	10 : 	(************* Check Sensors Before Homing ****************)
			Station.Status 		:= 'Org10: Check Sensors Before Homing';
			Station.StatusInt	:= 120;
			
			Station.OriginRunStep 	:= 20;	

	20	:	(********** Origin Condition Check ****************)
			IF  CO_FlapGuide_Cyl_Var.S_WorkPos AND CO_Brdg_Cyl_Var.S_WorkPos AND
				(H_ER_CtnRdyForPushIn AND NOT H_ER_CtnPushInDone) THEN
				Station.OriginRunStep 		:= Station.OriginRunStep + 10;				
			ELSE
				Station.OriginRunStep 		:= 100;
			END_IF
		
	30 : 	(************* Bridge Cylinder, Flap Guides Forward ****************)
		
			CO_Brdg_Cyl_Var.In_OrgWork 		:= TRUE;
			CO_Brdg_Cyl_Var.In_OrgHome 		:= FALSE;
			CO_FlapGuide_Cyl_Var.In_OrgWork := TRUE;
			CO_FlapGuide_Cyl_Var.In_OrgHome := FALSE;
			
			CO_YPush_Srv_Var.In_PosCmd := H_CO_YPush_Srv_CtnFinalPos;
			CO_YPush_Srv_Var.In_VelCmd := A_Srv_YPusherLoSpeed;
			IF CO_YPush_Srv_Var.In_MoveXLock AND CO_Brdg_Cyl_Var.In_WorkXLock THEN
				CO_YPush_Srv_Var.In_MoveAbs := TRUE;
			END_IF
		
			IF CO_Brdg_Cyl_Var.S_WorkPos AND 
				CO_FlapGuide_Cyl_Var.S_WorkPos THEN
				CO_YPush_Srv_Var.In_MoveAbs 		:= FALSE;
				CO_Brdg_Cyl_Var.In_AutoWork 		:= FALSE;
				CO_FFlapBrdg_Cyl_Var.In_OrgWork 	:= FALSE;
				CO_FlapGuide_Cyl_Var.In_OrgWork 	:= FALSE;
				Station.OriginRunStep  				:= Station.OriginRunStep  + 10;
			END_IF		
			
	40 : 	(************* Move Y Pusher To Push Stack into Carton  ****************)	
			CO_YPush_Srv_Var.In_PosCmd := H_CO_YPush_Srv_CtnFinalPos;
			CO_YPush_Srv_Var.In_VelCmd := A_Srv_YPusherLoSpeed;
			CO_YPush_Srv_Var.In_MoveAbs := TRUE;

			IF 	CO_YPush_Srv_Var.Out_CurrPos >= (CO_YPush_Srv_Var.In_PosCmd - 100) THEN
				CO_YPush_Strk_Cyl_Var.In_OrgWork := TRUE;
				CO_YPush_Strk_Cyl_Var.In_OrgHome := FALSE;
			END_IF
			
			IF ((fcComparePos(CurrPos:= CO_YPush_Srv_Var.Out_CurrPos, TargetPos:= CO_YPush_Srv_Var.In_PosCmd, Tolerance := 0.5)) AND
							CO_YPush_Srv_Var.Out_InPos) AND
				CO_YPush_Strk_Cyl_Var.S_WorkPos THEN	
				H_CO_StkRdyForYPush 				:= FALSE;	
				H_CO_Bdl_StkY_Count 				:= 0;	
				CO_YPush_Srv_Var.In_MoveAbs 		:= FALSE;
				CO_YPush_Strk_Cyl_Var.In_OrgWork 	:= FALSE;
				Station.OriginRunStep 				:= 50;
				
				IF NOT Cfg_BypassErector AND H_ER_CtnRdyForPushIn THEN
					H_ER_CtnPushInDone := TRUE;
				END_IF
					H_ER_CtnRdyForPushIn := FALSE;
				
			END_IF
			
	50 : 	(************* push into box  after y push  ****************)
			Station.Status 		:= '120: Push into box';
			Station.StatusInt	:= 151;
			
			CO_YPush_Cyl_Var.In_OrgWork := TRUE;
			CO_YPush_Cyl_Var.In_OrgHome := FALSE;
			
			IF  CO_YPush_Cyl_Var.S_HomePos THEN
				CO_YPush_Cyl_Var.In_AutoWork := TRUE;
				CO_YPush_Cyl_Var.In_AutoHome := FALSE;			
				CO_YPush_Srv_Var.In_MoveAbs := FALSE; 
				Station.RunStep := 100;			
			END_IF
			
	
			
	100 : 	(************* Y Pusher Servo Move to Safe Pos ****************)
			Station.Status 		:= 'Org30: Y Pusher Servo Move to Safe Pos ';
			Station.StatusInt	:= 172;
			CO_YPush_Strk_Cyl_Var.In_OrgHome 	:= NOT CO_YPush_Strk_Cyl_Var.S_HomePos;	
			
		IF CO_YPush_Srv_Var.Out_CurrPos > H_CO_YPush_Srv_SafePosition THEN
			CO_YPush_Srv_Var.In_PosCmd := H_CO_YPush_Srv_SafePosition; 
			CO_YPush_Srv_Var.In_VelCmd := A_Srv_BeltAutoHiSpeed;
			CO_YPush_Srv_Var.In_MoveAbs := TRUE;
		ELSE
			CO_YPush_Srv_Var.In_MoveAbs := FALSE;
			Station.OriginRunStep := Station.OriginRunStep+5;	
		END_IF
				
			IF ((fcComparePos(CurrPos:= CO_YPush_Srv_Var.Out_CurrPos, TargetPos:= H_CO_YPush_Srv_SafePosition,  Tolerance := 0.5)) AND
				CO_YPush_Srv_Var.Out_InPos) THEN
				CO_YPush_Srv_Var.In_MoveAbs := FALSE;
				Station.OriginRunStep := Station.OriginRunStep+5;	
			END_IF
			
	105:	(************* Y Pusher Servo Move to Standby Pos ****************)			
			CO_YPush_Cyl_Var.In_OrgWork := TRUE;
			CO_YPush_Cyl_Var.In_OrgHome := FALSE;
			
			IF CO_YPush_Cyl_Var.S_WorkPos THEN
				CO_YPush_Srv_Var.In_PosCmd := H_CO_YPush_Srv_CurrStandbyPos; 
				CO_YPush_Srv_Var.In_VelCmd := A_Srv_BeltAutoHiSpeed;
				CO_YPush_Srv_Var.In_MoveAbs := TRUE;
			END_IF
			
			IF ((fcComparePos(CurrPos:= CO_YPush_Srv_Var.Out_CurrPos, TargetPos:= H_CO_YPush_Srv_CurrStandbyPos, Tolerance := 0.5)) AND
							CO_YPush_Srv_Var.Out_InPos) THEN
				CO_YPush_Srv_Var.In_MoveAbs := FALSE;
			Station.OriginRunStep := Station.OriginRunStep+5;	
			END_IF
			
	110 : 	(************* All Cylinders Home ****************)
			Station.Status 		:= 'Org40: All Cylinders Home';
			Station.StatusInt	:= 173;
			
			
			CO_Brdg_Cyl_Var.In_OrgHome 			:= NOT CO_Brdg_Cyl_Var.S_HomePos;
			CO_Brdg_Cyl_Var.In_OrgWORK			:= FALSE;	
			CO_FlapGuide_Cyl_Var.In_OrgHome 	:= NOT CO_FlapGuide_Cyl_Var.S_HomePos;				
			CO_YPush_Cyl_Var.In_OrgWork 		:= FALSE;
			CO_YPush_Cyl_Var.In_OrgHome 		:= TRUE;


			IF  CO_YPush_Strk_Cyl_Var.S_HomePos AND
				CO_Brdg_Cyl_Var.S_HomePos 		AND
				CO_FlapGuide_Cyl_Var.S_HomePos 	AND
				CO_YPush_Cyl_Var.S_HomePos		THEN
				CO_YPush_Strk_Cyl_Var.In_OrgHome 	:= FALSE;	
				CO_Brdg_Cyl_Var.In_OrgHome 			:= FALSE;	
				CO_FlapGuide_Cyl_Var.In_OrgHome 	:= FALSE;
				CO_YPush_Cyl_Var.In_OrgWork 		:= FALSE;
				CO_YPush_Cyl_Var.In_OrgHome 		:= FALSE;

				IF CO_YPush_WA_Origin THEN
					Station.OriginRunStep := 0;	
				END_IF	
			END_IF
		


					
	END_CASE

ELSE

	Station.OriginRunStep := 0;	
	
END_IF

END_PROGRAM

// ---- POUs/Collator/CO_Cylinder_Output.TcPOU
PROGRAM CO_Cylinder_Output
VAR
	Reset:BOOL;
	bEnable:BOOL;
	CO_Brdg_Cyl_Home_Tmr : TON;
	CO_Brdg_Cyl_Work_Tmr : TON;
	
END_VAR

bEnable := NOT MC.Trouble;

(*Refer to FastTask Folder for Stack Release Cylinder Control*)

CO_Brdg_Cyl_Var.In_HomeXLock := TRUE;
CO_Brdg_Cyl_Var.In_WorkXLock := (NOT ER_Arm_Srv_Var.Out_Busy OR NOT ER_Arm_Vac_Var.S_Vacuum) AND
								ER_RFlapL_Cyl_Var.S_HomePos;
CO_Brdg_Cyl_Home_Tmr(IN:= O_CO_Brdg_Bwd, PT := T#2S);
CO_Brdg_Cyl_Work_Tmr(IN:= O_CO_Brdg_Fwd, PT := T#2S);

CO_Brdg_Cyl(				
	IN_CylName		:='3Y3 PUSHER BRIDGE', 	
	In_Enable		:= bEnable, 	
	In_Reset		:= MC.ResetPressed, 	
	In_WorkRS		:= I_CO_Brdg_Fwd, 	
	In_HomeRS		:= I_CO_Brdg_Bwd, 	
	In_WorkTON		:= T#10MS, 	
	In_HomeTON		:= T#10MS, 	
	in_Timeout		:= TP_Cyl_Timeout, 	
	Out_WorkSV		=> O_CO_Brdg_Fwd, 	
	Out_HomeSV		=> O_CO_Brdg_Bwd, 	
	CylVar			:= CO_Brdg_Cyl_Var,
	Station			:= SC[2]);

CO_FlapGuide_Cyl_Var.In_HomeXLock := TRUE;
CO_FlapGuide_Cyl_Var.In_WorkXLock := TRUE;

CO_FlapGuide_Cyl(				
	IN_CylName		:='3Y4/5 PUSHER FLAP GUIDE', 	
	In_Enable		:= bEnable, 	
	In_Reset		:= MC.ResetPressed, 	
	In_WorkRS		:= I_CO_RFlapGuide_Fwd AND I_CO_FFlapGuide_Fwd, 	
	In_HomeRS		:= I_CO_RFlapGuide_Bwd AND I_CO_FFlapGuide_Bwd, 	
	In_WorkTON		:= T#10MS, 	
	In_HomeTON		:= T#10MS, 	
	in_Timeout		:= TP_Cyl_Timeout, 	
	Out_WorkSV		=> O_CO_RFlapGuide_Fwd, 	
	Out_HomeSV		=> O_CO_RFlapGuide_Bwd, 	
	CylVar			:= CO_FlapGuide_Cyl_Var,
	Station			:= SC[2]);

	O_CO_FFlapBrdg_Fwd:=O_CO_RFlapGuide_Fwd;
	O_CO_FFlapBrdg_Bwd:=O_CO_RFlapGuide_Bwd;
	
CO_YPush_Strk_Cyl_Var.In_HomeXLock := TRUE;
CO_YPush_Strk_Cyl_Var.In_WorkXLock := CO_YPush_Cyl_Var.S_HomePos;

CO_YPush_Strk_Cyl(				
	IN_CylName		:='3Y2 Y PUSHER STROKE', 	
	In_Enable		:= bEnable, 	
	In_Reset		:= MC.ResetPressed, 	
	In_WorkRS		:= I_CO_YPush_Strk_Fwd, 	
	In_HomeRS		:= I_CO_YPush_Strk_Bwd, 	
	In_WorkTON		:= T#10MS, 	
	In_HomeTON		:= T#10MS, 	
	in_Timeout		:= TP_Cyl_Timeout, 	
	Out_WorkSV		=> O_CO_YPush_Strk_Fwd, 	
	Out_HomeSV		=> O_CO_YPush_Strk_Bwd, 	
	CylVar			:= CO_YPush_Strk_Cyl_Var,
	Station			:= SC[2]);

CO_YPush_Cyl_Var.In_HomeXLock := TRUE ;
CO_YPush_Cyl_Var.In_WorkXLock := CO_YPush_Srv_Var.Out_CurrPos <= H_CO_YPush_Srv_SafePosition + 1 ;

CO_YPush_Cyl(				
	IN_CylName		:='3Y1 Y PUSHER', 	
	In_Enable		:= bEnable, 	
	In_Reset		:= MC.ResetPressed, 	
	In_WorkRS		:= I_CO_YPush_Up, 	
	In_HomeRS		:= I_CO_YPush_Dn, 	
	In_WorkTON		:= T#10MS, 	
	In_HomeTON		:= T#10MS, 	
	in_Timeout		:= TP_Cyl_Timeout, 	
	Out_WorkSV		=> O_CO_YPush_Up, 	
	Out_HomeSV		=> O_CO_YPush_Dn, 	
	CylVar			:= CO_YPush_Cyl_Var,
Station			:= SC[2]);

CO_PalletLoc_Cyl_Var.In_HomeXLock := TRUE;
CO_PalletLoc_Cyl_Var.In_WorkXLock := TRUE;
	
CO_PalletLoc_Cyl(				
	IN_CylName		:='3Y2 Y PALLET LOCATING', 	
	In_Enable		:= bEnable, 	
	In_Reset		:= MC.ResetPressed, 	
	In_WorkRS		:= I_CO_PalletLocating_Fwd, 	
	In_HomeRS		:= I_CO_PalletLocating_Bwd, 	
	In_WorkTON		:= T#10MS, 	
	In_HomeTON		:= T#10MS, 	
	in_Timeout		:= TP_Cyl_Timeout, 	
	Out_WorkSV		=> O_CO_PalletLocating_Fwd, 	
	Out_HomeSV		=> O_CO_PalletLocating_Bwd, 	
	CylVar			:= CO_PalletLoc_Cyl_Var,
	Station			:= SC[2]);

CO_Sing1_Cyl_Var.In_HomeXLock := TRUE;
CO_Sing1_Cyl_Var.In_WorkXLock := TRUE;
CO_Sing1_Cyl(				
	IN_CylName		:='3Y2 Singulator 1', 	
	In_Enable		:= bEnable, 	
	In_Reset		:= MC.ResetPressed, 	
	In_WorkRS		:= I_CO_Sing1_Fwd, 	
	In_HomeRS		:= I_CO_Sing1_Bwd, 	
	In_WorkTON		:= T#10MS, 	
	In_HomeTON		:= T#10MS, 	
	in_Timeout		:= TP_Cyl_Timeout, 	
	Out_WorkSV		=> O_CO_Sing1_Fwd, 	
	Out_HomeSV		=> O_CO_Sing1_Bwd, 	
	CylVar			:= CO_Sing1_Cyl_Var,
	Station			:= SC[2]);

CO_Sing2_Cyl_Var.In_HomeXLock := TRUE;
CO_Sing2_Cyl_Var.In_WorkXLock := TRUE;	
CO_Sing2_Cyl(				
	IN_CylName		:='3Y2 Singulator 1', 	
	In_Enable		:= bEnable, 	
	In_Reset		:= MC.ResetPressed, 	
	In_WorkRS		:= I_CO_Sing2_Fwd, 	
	In_HomeRS		:= I_CO_Sing2_Bwd, 	
	In_WorkTON		:= T#10MS, 	
	In_HomeTON		:= T#10MS, 	
	in_Timeout		:= TP_Cyl_Timeout, 	
	Out_WorkSV		=> O_CO_Sing2_Fwd, 	
	Out_HomeSV		=> O_CO_Sing2_Bwd, 	
	CylVar			:= CO_Sing2_Cyl_Var,
	Station			:= SC[2]);

END_PROGRAM

// ---- POUs/Collator/CO_Servo_Output.TcPOU
PROGRAM CO_Servo_Output
VAR
	Reset:BOOL;
	plsStopMove: R_trig;
	bEnable: BOOL;
	bEnable_Stack: BOOL;
	bEnable_XPush: BOOL;
	bEnable_YPush: BOOL;
END_VAR

IF (MC.AutoMode OR SC[1].M_Step OR SC[2].M_Step) AND NOT CO.Bypass THEN
	CO_YPush_Srv_Var.In_ServoOn := TRUE;
END_IF

IF CO.OriginSchRun OR MC.OriginSchRun or mc.AutoMode or (mc.ResetPressed AND NOT mc.Trouble) THEN
	CO_YPush_Srv_Var.In_ServoOn := TRUE;
END_IF

 
bEnable_Stack := NOT (CO_Stack.MajorFault OR CO_Stack.MinorFault OR CO_Stack.DeviceFault OR MC.Trouble);
bEnable_YPush := NOT (CO_YPush.MajorFault OR CO_YPush.MinorFault OR CO_YPush.DeviceFault OR MC.Trouble);


(*CO_M5 Collator Y Pusher Motor - 111M1*)

IF Cfg_CollDircLtoR THEN
CO_YPush_Srv_Var.In_MoveXLock := 	((CO_FlapGuide_Cyl_Var.S_WorkPos AND
										ER_FFlapL_Cyl_Var.S_HomePos AND
										ER_RFlapL_Cyl_Var.S_HomePos) OR
									(CO_YPush_Srv_Var.Out_CurrPos <= H_CO_YPush_Srv_CtnFinalPos+200)) ;
ELSE
CO_YPush_Srv_Var.In_MoveXLock := 	((CO_FlapGuide_Cyl_Var.S_WorkPos AND
										ER_FFlapR_Cyl_Var.S_HomePos AND
										ER_RFlapR_Cyl_Var.S_HomePos) OR
									(CO_YPush_Srv_Var.Out_CurrPos <= H_CO_YPush_Srv_CtnFinalPos+200));
END_IF
CO_YPush_Srv_Drive(
	In_Enable:= bEnable_YPush, 
	In_Reset := MC.ResetPressed,
	In_AbsEncoder:= TRUE, 
	In_DriveInput:= CO_YPush_Srv_Input, 
	In_CommState:= CO_YPush_Srv_State, 
	Out_DriveOutput=> CO_YPush_Srv_Output, 
	Out_DriveFeedRateOverride=> CO_YPush_Srv_Feedrate, 
	DriveVar:= CO_YPush_Srv_Var,
	Station			:= SC[2]);

IF mc.ManualMode THEN	
	CO_YPush_Srv_Feedrate := 10000;
ELSE
	CO_YPush_Srv_Feedrate :=    INT_TO_UINT(hmi.V_MachineSpeed * 100);
END_IF

END_PROGRAM

// ---- POUs/Collator/CO_Nordson.TcPOU
PROGRAM CO_Nordson
VAR
	PumpOnOff	: fbOnOffDevCtrl;
	Standby		: fbOnOffDevCtrl;
	HeaterOn	: fbOnOffDevCtrl;
END_VAR



PumpOnOff(
	IN_DevName:= 'Pump OnOff', 
	In_Enable:= TRUE, 
	In_Reset:= MC.ResetPressed, 
	In_AutoON:= ER_Nordson_PumpOnOff_Var.In_AutoON , 
	In_OrgON:= ER_Nordson_PumpOnOff_Var.In_OrgOn , 
	In_OnXLock:= TRUE, 
	In_ONSig:=PumpOnOff.Out_OnSV , 
	In_OnTON:= , 
	in_Timeout:= T#1S, 
	Out_OnSV=> O_Nord_Auto , 
	E_OnErr=> , 
	S_OnSig=> );
	
Standby(
	IN_DevName:= 'Standby', 
	In_Enable:= TRUE, 
	In_Reset:= MC.ResetPressed, 
	In_AutoON:= ER_Nordson_Standby_Var.In_AutoON , 
	In_OrgON:= ER_Nordson_Standby_Var.In_OrgOn, 
	In_OnXLock:= TRUE , 
	In_ONSig:= Standby.Out_OnSV, 
	In_OnTON:= , 
	in_Timeout:= T#1S, 
	Out_OnSV=> O_Nord_Standby , 
	E_OnErr=> , 
	S_OnSig=> );	
	
HeaterOn(
	IN_DevName:= 'Heater On', 
	In_Enable:= TRUE, 
	In_Reset:= MC.ResetPressed, 
	In_AutoON:= ER_Nordson_HeaterOn_Var.In_AutoON  , 
	In_OrgON:= ER_Nordson_HeaterOn_Var.In_OrgOn, 
	In_OnXLock:= TRUE , 
	In_ONSig:= HeaterOn.Out_OnSV, 
	In_OnTON:= , 
	in_Timeout:= T#1S, 
	Out_OnSV=> O_Nord_HeaterOn , 
	E_OnErr=> , 
	S_OnSig=> );

END_PROGRAM

// ---- POUs/FB/fbOnOffDevCtrl.TcPOU
FUNCTION_BLOCK fbOnOffDevCtrl

VAR_INPUT
	IN:BOOL;
	IN_DevName:STRING;
	In_Enable:BOOL;
	In_Reset:BOOL;


	(*Trigger*)
	In_AutoON:BOOL;
	In_OrgON:BOOL;

	(*Mechanical Interlock*)
	In_OnXLock:BOOL;

	(*Sensors*)
	In_ONSig:BOOL;

	(*Timer*)
	In_OnTON:TIME;
	in_Timeout:TIME;

END_VAR

VAR_OUTPUT
	Q:BOOL;
	Out_OnSV:BOOL;
	E_OnErr:BOOL;
	S_OnSig:BOOL;

END_VAR

VAR_IN_OUT
	
END_VAR

VAR

	(* Trigger*)
	T_ManOn:BOOL;
	T_ManOff:BOOL;

	Loc_On:BOOL;
	On_TOut: TON;
	On_TON: TON;
	Loc_OnPls: BOOL;
	OnPls: R_TRIG;
	Out_RSErr:BOOL;
	OnPosPls: F_TRIG;

END_VAR
VAR_IN_OUT

END_VAR
VAR // added by the converter: edge detectors and wires of the graphical bodies
    _w1 : BOOL;
END_VAR

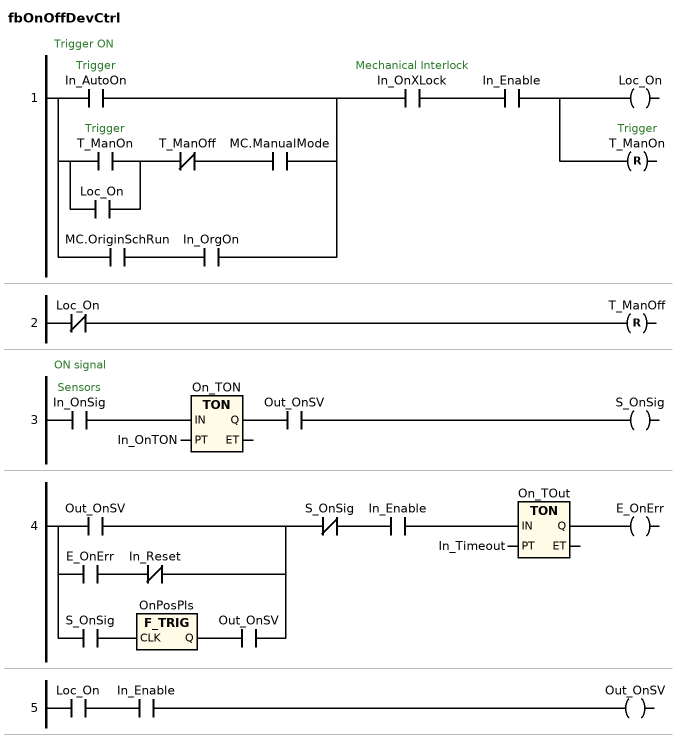
// NETWORK 1
// Trigger ON
//   In_AutoOn: Trigger
//   T_ManOn: Trigger
//   In_OnXLock: Mechanical Interlock
_w1 := (In_AutoOn OR (T_ManOn OR Loc_On) AND NOT T_ManOff AND MC.ManualMode OR MC.OriginSchRun AND In_OrgOn) AND In_OnXLock AND In_Enable;
Loc_On := _w1;
T_ManOn R= _w1;

// NETWORK 2
T_ManOff R= NOT Loc_On;

// NETWORK 3
// ON signal
//   In_OnSig: Sensors
//   In_OnTON: Timer
On_TON(IN := In_OnSig, PT := In_OnTON); // TON
S_OnSig := On_TON.Q AND Out_OnSV;

// NETWORK 4
OnPosPls(CLK := S_OnSig); // F_TRIG
On_TOut(IN := (Out_OnSV OR E_OnErr AND NOT In_Reset OR OnPosPls.Q AND Out_OnSV) AND NOT S_OnSig AND In_Enable, PT := In_Timeout); // TON
E_OnErr := On_TOut.Q;

// NETWORK 5
Out_OnSV := Loc_On AND In_Enable;

END_FUNCTION_BLOCK

// ---- POUs/Erector/ER_Main.TcPOU
PROGRAM ER_Main
VAR
END_VAR

IF Cfg_BypassErector THEN
	HMI.T_Station_BypassP[3] := TRUE;
ELSE
	HMI.T_Station_BypassP[3] := FALSE;
END_IF

ER_Timers();

ER_Error			(Station:= SC[3]);
ER_Auto_Arm			(Station:= SC[3]);
ER_Auto_FixedFlap	(Station:= SC[3]);
ER_Glue				(Station:= SC[3]);
ER_Origin			(Station:= SC[3]);

ER_Cylinder_Output();
ER_Servo_Output();
ER_Motor_Output();
ER_Vacuum_Output();

(* ER Structure is only for displaying on HMI*)
SC[3].T_OriginSearch := ER.T_OriginSearch;
ER := SC[3];

(*debug*)

IF T_SimPushIn THEN
	H_ER_CtnRdyForPushIn := FALSE;
	H_ER_CtnPushInDone := TRUE;
	H_ER_CtnSideFlapDone := FALSE;
END_IF

END_PROGRAM

// ---- POUs/Erector/ER_Timers.TcPOU
PROGRAM ER_Timers
VAR
	ER_Carton_TON	:ton;
	
END_VAR


ER_BufCv_Ctn_TON 	(IN := 	I_ER_RefillL_PE AND 
							I_ER_EmptyL_PE	AND
							I_ER_EmptyR_PE	AND
							I_ER_BufferL_PE	AND
							I_ER_BufferR_PE, pt := T#0.5S);
ER_Carton_TON(IN := 		I_ER_EmptyL_PE	AND
							I_ER_EmptyR_PE	AND
							I_ER_BufferL_PE	AND
							I_ER_BufferR_PE, pt := T#1S); 
							
ER_BufCvL_Ctn_TON 	(IN := (I_ER_EmptyL_PE AND mc.AutoRunning) OR I_ER_BufferL_PE , pt := T#70MS);
ER_BufCvR_Ctn_TON 	(IN := (I_ER_EmptyR_PE AND mc.AutoRunning) OR I_ER_BufferR_PE , pt := T#70MS);

END_PROGRAM

// ---- POUs/Erector/ER_Error.TcPOU
PROGRAM ER_Error
VAR_IN_OUT
	Station		:structStationCtrl;
END_VAR

VAR
	CaseBufferWaitTON			:Ton;
	CaseBufferEmpty_ResetTON	:ton;
	GlueEmpty_ResetTON			:ton;
	CaseBufferEmptySen_Timeout	:ton;

END_VAR

IF MC.ResetPressed THEN
	Station.SeqFaultWord := 0;
END_IF

(* 	Reserved Station.SeqFaultWord 
	= 1~49 for Major Fault
	= 100~149 for Origin Sequence Fault
	= 150~199 for Origin Width Adjust Sequence Fault
	= 200~299 for Auto Sequence Fault
	= 300~399 for misc fault listed on this page*)

Station.MajorFault := ((Station.SeqFaultWord > 0) 	AND (Station.SeqFaultWord < 50)) OR E_Case_Infeed_Safety_NOk ;
Station.MinorFault := (Station.SeqFaultWord >= 100) OR Station.DeviceFault 
													OR E_Nordson_Alarm 
													OR E_CaseBufferAlignment_Err
													OR ((E_ER_EmptyL_PE
													OR E_ER_BufferL_PE
													OR E_ER_EmptyR_PE
													OR E_ER_BufferR_PE) AND sc[3].RunStep = 0);
									
													
(* Case Infeed safety not OK *)
IF NOT I_Case_Infeed_Safety_Ok AND I_Emg_SC_OK AND I_Door_SC_OK AND NOT MC_WA_Run AND NOT Erector_SafetySensorBypass THEN
	E_Case_Infeed_Safety_NOk	:= TRUE;
END_IF

(* Case Buffer Error *)
CaseBufferWaitTON			(IN:= ((I_ER_EmptyL_PE AND NOT I_ER_BufferL_PE) OR (I_ER_EmptyR_PE AND NOT I_ER_BufferR_PE)) AND mc.AutoRunning AND (sc[3].RunStep = 0), PT:= T#30S); 
IF CaseBufferWaitTON.Q THEN
	E_CaseBufferAlignment_Err	:= TRUE;
END_IF
(*
W_CaseBuffer_is_Empty	:= 	(CaseBufferEmptying_Counter >= CaseBufferEmptying_Setting);
CaseBufferEmpty_ResetTON	( IN:= I_ER_RefillL_PE, pt:= T#3S);
IF CaseBufferEmpty_ResetTON.Q THEN
	CaseBufferEmptying_Counter	:= 0;
END_IF
*)
CaseBufferEmptySen_Timeout	( IN:= (I_ER_EmptyL_PE AND NOT I_ER_EmptyR_PE) OR (I_ER_EmptyR_PE AND NOT I_ER_EmptyL_PE), pt:= T#10S);
IF CaseBufferEmptySen_Timeout.Q THEN
	E_CaseBuffer_EmptySensors	:= TRUE;
END_IF


(*Refill Carton Buffer Warning*)
W_ER_BufRefill		:= MC.AutoMode AND NOT Station.Bypass AND 
						NOT I_ER_RefillL_PE AND NOT HMI.T_EndProd;



(* Glue Alarm/Warning *)
(*E_Nordson_Alarm		:= (NOT I_Nord_Rdy AND T_GlueEnable) AND NOT mc.DryRun AND mc.AutoRunning;*)
W_Glue_Low_Level	:= I_Nord_TankLow;
W_Glue_is_Empty		:= (GlueEmptying_Counter >= GlueEmptying_Setting );
IF NOT I_Nord_TankLow THEN 
	GlueEmptying_Counter	:= 0;
END_IF

END_PROGRAM

// ---- POUs/Erector/ER_Auto_Arm.TcPOU
                                                                                                                                                                                                                                                                                                      PROGRAM ER_Auto_Arm
VAR_IN_OUT
	Station		:structStationCtrl;
END_VAR
VAR
	tmrDelayBFlapUp:ton;
	Timeout					:TON;	
	StpCtnPE_TOFF			:Ton;
	ManualInit_TOn			:Ton;
	tmrDelayVacHold			:ton;
	CaseSupply_L_Timeout	:TON;
	CaseSupply_R_Timeout	:TON;
	tmr_Case_Buffer			:ton;	
	tmr_ArmTiltDly			:Ton;
	ServoTargetPos			:REAL;
	TimeoutTrigger			:BOOL;
	TimeoutSetting			:TIME;
	NoWPonErector			:BOOL;
	NoWPonExit				:BOOL;
	CartonPreAtStopper		:BOOL;
	GlueStart1 				:BOOL;
	GlueStart2 				:BOOL;
	DistanceAdvanceForGlue	:REAL;
	End_Production			:BOOL;	
	Case_Not_Ready 			:BOOL;	
	CaseSupply_L_TimeoutM	:BOOL;
	CaseSupply_R_TimeoutM	:BOOL;
			
END_VAR

NoWPonErector := 	NOT H_ER_CtnRdyForPushIn AND 
					NOT I_ER_StpL_Ctn_PE AND
					NOT I_ER_StpR_Ctn_PE;
							
NoWPonExit := 	NOT H_ER_CtnRdyForGlue AND
				NOT H_ER_CtnGlueDone AND
				NOT I_EX_Cv_Ctn_PE;

tmr_Case_Buffer	(IN := NOT ER_BufCv_Ctn_TON.Q AND 
					NOT (MC.DryRun  OR  End_Production ) AND
					mc.AutoRunning, pt := T#3S);			
Case_Not_Ready := 	(tmr_Case_Buffer.Q AND NOT mc.DryRun) OR 
					(NOT I_Case_Infeed_Safety_Ok AND NOT mc.E_EmgStop AND NOT mc.E_SafetyDoorOpen);
					
					
sc[3].Warning			:= Case_Not_Ready;
				
(**************************************************************************************************************)
(*	Initial Device	*)
(**************************************************************************************************************)
ManualInit_TOn (in:= mc.ManualMode AND NOT mc.OriginSchRun, pt:= T#1S);

IF mc.ManualMode AND NOT mc.OriginSchRun AND NOT ManualInit_TOn.Q THEN
	ER_Arm_Srv_Var.In_MoveAbs 			:= FALSE;
	ER_WA_Srv_Var.In_MoveAbs 			:= FALSE;	
	EX_HeightL_WA_Srv_Var.In_MoveAbs	:= FALSE;
	EX_HeightR_WA_Srv_Var.In_MoveAbs	:= FALSE;
END_IF
				
(**************************************************************************************************************)
(* GENERAL STATION MAPPING  *)
(**************************************************************************************************************)
Station.Name			:=	'CARTON ERECTOR & SIDE FLAP CLOSING';
Station.Rdy 			:= 	Station.Origin AND ER_Origin.ER_WA_Origin;
Station.AutoRun 		:=	(MC.AutoRunning OR Station.M_Step) AND 
							NOT (Station.Bypass OR Station.MajorFault OR Station.MinorFault);
Station.RunReq			:= 	(
							((NOT I_EX_Cv_Ctn_PE OR NoWPonErector) AND NoWPonErector AND NOT End_Production ) OR
							(H_ER_CtnSideFlapDone AND NoWPonExit)
							) AND
							(er_tIMERS.ER_Carton_TON.Q OR MC.DryRun OR 
							(End_Production AND (I_ER_StpL_Ctn_PE OR I_ER_StpR_Ctn_PE)) 
							);											
Station.RunCond			:=	(NOT CO_YPush.Running OR CO_YPush.RunStep >= 200) AND	(*Y Pusher Not Running Forward*) 
							( (I_Nord_Rdy and not W_Glue_is_Empty and not W_CaseBuffer_is_Empty)  OR NOT T_GlueEnable OR mc.DryRun) AND
							((NOT EX.Running OR										(*Hot Glue and Weight Check Not Running*) 	
							NoWPonErector)) AND
							NOT Station.Running AND									(*Fixed Flap Closing Not Running*)
							NOT (Station.Done OR MC.StopPressed);
Station.Run_NextStepPls	:=	(Station.AutoRun AND NOT Station.M_Step) OR 
							(Station.M_Step AND M_StepFwdPls) OR HMI.T_OneCycleRun;
Station.Run_PrevStepPls	:=	(Station.M_Step AND M_StepBwdPls);

(**************************************************************************************************************)
(* Auto Sequance*)
(**************************************************************************************************************)

Timeout(IN:=TimeoutTrigger, PT:=TimeoutSetting);
IF Timeout.Q THEN
	TimeoutTrigger := FALSE;
END_IF


tmrDelayVacHold	(IN:=Station.RunStep=30, PT:=T#0S);
tmr_ArmTiltDly	(IN:=Station.RunStep=20 AND ER_ArmTilt_Cyl_Var.S_HomePos, pt:= T#0.2S);
 
(********************* Case Supply Sequence Start ********************************)
	CaseSupply_L_Timeout	(IN:= ER_BufCvL_Mtr_Var.S_Running, PT:= T#60S);
	CaseSupply_R_Timeout	(IN:= ER_BufCvR_Mtr_Var.S_Running, PT:= T#60S);
	
	IF CaseSupply_L_Timeout.q THEN
		CaseSupply_L_TimeoutM	:= TRUE;
	END_IF
	IF CaseSupply_R_Timeout.q THEN
		CaseSupply_R_TimeoutM	:= TRUE;
	END_IF
	IF I_ER_RefillL_PE OR NOT mc.AutoRunning THEN
		CaseSupply_L_TimeoutM	:= FALSE;
		CaseSupply_R_TimeoutM	:= FALSE;
	END_IF
		
	ER_BufCvL_Mtr_Var.In_AutoON := NOT  ER_BufCvL_Ctn_TON.Q AND NOT CaseSupply_L_TimeoutM AND NOT(STation.RunStep >= 20 AND Station.RunStep <40)  ;
	ER_BufCvR_Mtr_Var.In_AutoON := NOT  ER_BufCvR_Ctn_TON.Q AND	NOT CaseSupply_L_TimeoutM AND NOT(STation.RunStep >= 20 AND Station.RunStep <40)  ;	


IF Station.AutoRun OR Station.M_Step THEN

(**************************************************************************)
	CASE Station.RunStep OF

	0 : 	(************* Ready To Run ****************)
			End_Production := hmi.T_EndProd;
			
			IF Station.RunCond AND Station.RunReq AND Station.Rdy  AND
				(NOT H_ER_CtnPushInDone OR H_ER_CtnSideFlapDone)  THEN
				Station.RunStep := Station.RunStep + 5;
			ELSIF NOT Station.RunCond THEN
				Station.Status 		:= '0: Station Waiting for Run Conditions';
				Station.StatusInt	:= 1;
			ELSIF NOT Station.RunReq THEN
				Station.Status 		:= '0: Station Waiting for Run Request';
				Station.StatusInt	:= 2;
			ELSE
				Station.Status 		:= '0: Station Not Ready';
				Station.StatusInt	:= 3;
			END_IF

	5 : 	(************* Stopper Down ****************)
			(************* Case Guide Down ****************)
			Station.Status 		:= '5: Stopper & Case Guide Down';
			Station.StatusInt	:= 251;
			
			ER_StpR_Cyl_Var.In_AutoWork 		:= FALSE;
			ER_StpR_Cyl_Var.In_AutoHome 		:= TRUE;
			ER_StpL_Cyl_Var.In_AutoWork 		:= FALSE;
			ER_StpL_Cyl_Var.In_AutoHome 		:= TRUE;
			ER_CaseGuideL_Cyl_Var.In_AutoWork 	:= FALSE;
			ER_CaseGuideL_Cyl_Var.In_AutoHome 	:= TRUE;
			ER_CaseGuideR_Cyl_Var.In_AutoWork 	:= FALSE;
			ER_CaseGuideR_Cyl_Var.In_AutoHome 	:= TRUE;
			

			IF 	ER_StpR_Cyl_Var.S_HomePos AND 
				ER_StpL_Cyl_Var.S_HomePos AND
				ER_CaseGuideL_Cyl_Var.S_HomePos AND
				ER_CaseGuideR_Cyl_Var.S_HomePos AND
				Station.Run_NextStepPls THEN
				ER_StpR_Cyl_Var.In_AutoWork := FALSE;
				ER_StpL_Cyl_Var.In_AutoWork := FALSE;
				H_ER_CtnErected				:= FALSE;
				IF NOT End_Production THEN
					Station.RunStep := Station.RunStep + 5;	
				ELSE
					Station.RunStep := 30;
				END_IF
			END_IF
			
	10 : 	(************* Erector Arm Servo Move forward while Vacuum ON ****************)
			Station.Status 		:= '10: Erector Arm Servo Move Forward';
			Station.StatusInt	:= 252;
			
			IF NOT MC.DryRun  THEN
				ER_Arm_Vac_Var.In_AutoVacuum := TRUE;
				ER_Arm_Vac_Var.In_AutoPurge := FALSE;
			END_IF

			ER_Arm_Srv_Var.In_PosCmd := H_ER_Arm_Srv_CtnVacuumPos + 45;
			ER_Arm_Srv_Var.In_VelCmd := A_Srv_ErectorArmHiSpeed;
			ER_Arm_Srv_Var.In_MoveAbs := TRUE;
			
			IF H_ER_CtnSideFlapDone THEN
				ER_RFlapL_Cyl_Var.In_AutoWork := TRUE;
				ER_RFlapR_Cyl_Var.In_AutoWork := TRUE;
			END_IF
			
			IF fcComparePos(CurrPos:= ER_Arm_Srv_Var.Out_CurrPos, TargetPos:= ER_Arm_Srv_Var.In_PosCmd,5) AND
				((ER_RFlapL_Cyl_Var.S_WorkPos AND ER_RFlapR_Cyl_Var.S_WorkPos) OR
					NOT H_ER_CtnSideFlapDone) AND
					(ER_Arm_Vac_Var.S_Vacuum OR MC.DryRun) AND
				Station.Run_NextStepPls THEN				
				ER_Arm_Srv_Var.In_MoveAbs := FALSE;
				ER_Arm_Vac_Var.In_AutoVacuum := FALSE;
				Station.RunStep := Station.RunStep + 10;	
			END_IF
	
	20 : 	(************* Erector Arm Servo Move backwards to pull out carton at slower speed ****************)
			(************* Rear Flap Close And Top Flap Close Home ****************)
			Station.Status 		:= '20: Erector Arm Servo Move Backwards to Pull Out Carton';
			Station.StatusInt	:= 253;
	
				ER_ArmTilt_Cyl_Var.In_AutoHome 	:= TRUE;
				ER_ArmTilt_Cyl_Var.In_AutoWork 	:= FALSE;
				
				H_HOR_CtnWeightOK				:= FALSE;				

				ServoTargetPos := H_ER_Arm_Srv_CtnVacuumPos - 100;
				ER_Arm_Srv_Var.In_PosCmd := ServoTargetPos;
				ER_Arm_Srv_Var.In_VelCmd := A_Srv_ErectorArmLoSpeed;
			
			IF ER_ArmTilt_Cyl_Var.S_HomePos AND tmr_ArmTiltDly.Q THEN
				ER_Arm_Srv_Var.In_MoveAbs := TRUE;
			END_IF
				
			IF ER_Arm_Srv_Var.Out_Busy THEN
				ER_Arm_Srv_Var.In_MoveAbs := FALSE;
			END_IF
			
			IF (ER_Arm_Srv_Var.Out_CurrPos <= ServoTargetPos + 5) THEN	
				H_ER_CtnErected						:= TRUE;			
				ER_Arm_Srv_Var.In_MoveAbs 			:= FALSE;
				ER_RFlapL_Cyl_Var.In_AutoWork 		:= FALSE;
				ER_RFlapL_Cyl_Var.In_AutoHome 		:= TRUE;
				ER_RFlapR_Cyl_Var.In_AutoWork 		:= FALSE;
				ER_RFlapR_Cyl_Var.In_AutoHome 		:= TRUE;				
				Station.RunStep := Station.RunStep + 10;	
			END_IF

	30 : 	(************* Erector Arm Servo Move to Carton Erect Final Position and Cylinders Bwd ****************)
			Station.Status 		:= '30: Erector Arm Servo Move to Carton Erect Final Position';
			Station.StatusInt	:= 254;
			
			ER_Arm_Srv_Var.In_PosCmd := H_ER_Arm_Srv_CtnErectPos;
			ER_Arm_Srv_Var.In_VelCmd := A_Srv_ErectorArmHiSpeed ;
			ER_Arm_Srv_Var.In_MoveAbs := TRUE;
						
			StpCtnPE_TOFF(IN:= NOT (I_ER_StpL_Ctn_PE OR I_ER_StpR_Ctn_PE), PT:=T#0S);
			
			IF StpCtnPE_TOFF.Q AND 
				ER_Arm_Srv_Var.Out_CurrPos <= (H_ER_Arm_Srv_CtnErectPos + 200) THEN
				ER_ArmTilt_Cyl_Var.In_AutoHome 	:= TRUE;
				ER_ArmTilt_Cyl_Var.In_AutoWork 	:= FALSE;
			END_IF
			
			IF 	ER_Arm_Srv_Var.Out_CurrPos <= (H_ER_Arm_Srv_CtnErectPos + 200) AND
				NOT End_Production THEN
				ER_StpR_Cyl_Var.In_AutoWork 	:= TRUE;
				ER_StpR_Cyl_Var.In_AutoHome 	:= FALSE;
				ER_StpL_Cyl_Var.In_AutoWork 	:= TRUE;
				ER_StpL_Cyl_Var.In_AutoHome 	:= FALSE;
		
	
			END_IF			
			
			IF ER_Arm_Srv_Var.Out_CurrPos <= (H_ER_Arm_Srv_CtnVacuumPos - 300) THEN	
				ER_TFlapClsL_Cyl_Var.In_AutoWork	:= FALSE;
				ER_TFlapClsL_Cyl_Var.In_AutoHome	:= TRUE;
				ER_TFlapClsR_Cyl_Var.In_AutoWork	:= FALSE;
				ER_TFlapClsR_Cyl_Var.In_AutoHome	:= TRUE;	
			END_IF
			
			IF NOT Station.M_Step AND H_ER_CtnSideFlapDone  THEN
				H_ER_CtnRdyForGlue := TRUE;
			END_IF
			
			IF ER_Arm_Srv_Var.Out_CurrPos <= (H_ER_Arm_Srv_CtnVacuumPos - 100) THEN
				ER_RFlapL_Cyl_Var.In_AutoHome 		:= TRUE;
				ER_RFlapL_Cyl_Var.In_AutoWork 		:= FALSE;
				ER_RFlapR_Cyl_Var.In_AutoHome 		:= TRUE;
				ER_RFlapR_Cyl_Var.In_AutoWork 		:= FALSE;
				ER_BFlapCloseL_Cyl_Var.In_AutoHome 	:= TRUE;
				ER_BFlapCloseL_Cyl_Var.In_AutoWork	:= FALSE;
				ER_BFlapCloseR_Cyl_Var.In_AutoHome 	:= TRUE;
				ER_BFlapCloseR_Cyl_Var.In_AutoWork 	:= FALSE;
			END_IF
			
			IF fcComparePos(CurrPos:= ER_Arm_Srv_Var.Out_CurrPos, TargetPos:= ER_Arm_Srv_Var.In_PosCmd,3) THEN
				IF H_ER_CtnSideFlapDone THEN
					H_ER_CtnSideFlapDone 	:= FALSE;
					H_ER_CtnPushInDone 		:= FALSE;					
				END_IF
			END_IF
					
			IF fcComparePos(CurrPos:= ER_Arm_Srv_Var.Out_CurrPos, TargetPos:= ER_Arm_Srv_Var.In_PosCmd,3) AND
				ER_Arm_Srv_Var.Out_InPos AND
				ER_ArmTilt_Cyl_Var.S_HomePos AND
				ER_RFlapL_Cyl_Var.S_HomePos AND
				ER_RFlapR_Cyl_Var.S_HomePos AND
				tmrDelayVacHold.Q AND
				Station.Run_NextStepPls THEN		
				ER_StpR_Cyl_Var.In_AutoWork := FALSE;
				ER_StpL_Cyl_Var.In_AutoWork := FALSE;		
				ER_Arm_Srv_Var.In_MoveAbs := FALSE;
				ER_Arm_Cyl_Var.In_AutoWork := FALSE;
				ER_ArmTilt_Cyl_Var.In_AutoHome := FALSE;
				ER_BFlapCloseL_Cyl_Var.In_AutoHome := FALSE;
				ER_BFlapCloseR_Cyl_Var.In_AutoHome := FALSE;
	
				IF NOT (ER_StpR_Cyl_Var.S_WorkPos AND ER_StpL_Cyl_Var.S_WorkPos)AND 
					ER_Arm_Vac_Var.S_Vacuum AND NOT End_Production AND
					NOT MC.DryRun THEN
					Station.SeqFaultWord 		:= 200;	
					E_NoGapAtStoper				:= TRUE;		
					Station.SeqFaultString 		:= 'Auto: Stopper Sensor Did not Detect Gap between Carton';	
				ELSIF NOT (I_ER_StpL_Ctn_PE AND I_ER_StpR_Ctn_PE) AND
					NOT (MC.DryRun OR End_Production)  THEN 	
					Station.SeqFaultWord 		:= 104;
					Station.SeqFaultString 		:= 'Auto: Carton Missing or Not Properly Erected. Check Carton.';
					E_CaseNotDetected			:= TRUE;
				ELSIF NOT I_ER_StpL_Ctn_PE AND
					NOT (MC.DryRun OR End_Production)  THEN
					Station.SeqFaultWord 		:= 201;	
					E_LeftStopper_NotDetect		:= TRUE;
					Station.SeqFaultString 		:= 'Auto: Carton Not Detected by Left Stopper Sensor';				
				ELSIF NOT I_ER_StpR_Ctn_PE AND
					NOT (MC.DryRun OR End_Production) THEN
					Station.SeqFaultWord 		:= 202;
					E_RightStopper_NotDetect	:= TRUE;			
					Station.SeqFaultString 		:= 'Auto: Carton Not Detected by Right Stopper Sensor';			
				ELSE
					IF NOT End_Production  THEN
						Station.RunStep := Station.RunStep + 10;	
					ELSE
						Station.RunStep := 100;
					END_IF					
				END_IF
			END_IF
	35:		(* Erector Empty Carton sensor Off detection *)	
				IF I_ER_EmptyL_PE				THEN
					E_ER_EmptyL_PE	:=TRUE;
				ELSIF I_ER_BufferL_PE			THEN
					E_ER_BufferL_PE	:= TRUE;
				ELSIF I_ER_EmptyR_PE			THEN
					E_ER_EmptyR_PE	:= TRUE;
				ELSIF I_ER_BufferR_PE			THEN
					E_ER_BufferR_PE	:=TRUE;
				END_IF	
					Station.RunStep := Station.RunStep + 5;	
	
	40 : 	(************* Bottom Flap Holder Cyl Up & Vacuum ON ****************)
			(************* Case Guide Cyl Up  ****************)
			(************* Top Cyl Open  ****************)
			Station.Status 		:= '40: Bottom Flap Holder Cyl Up & Vacuum ON';
			Station.StatusInt	:= 255;



	
						
			IF	ER_CaseGuideL_Cyl_Var.S_WorkPos AND
				ER_CaseGuideR_Cyl_Var.S_WorkPos THEN						
				ER_BFlapL_Cyl_Var.In_AutoWork 		:= TRUE;
				ER_BFlapL_Cyl_Var.In_AutoHome 		:= FALSE;
				ER_BFlapR_Cyl_Var.In_AutoWork 		:= TRUE;
				ER_BFlapR_Cyl_Var.In_AutoHome 		:= FALSE;
			END_IF
			ER_CaseGuideL_Cyl_Var.In_AutoWork	:= TRUE;
			ER_CaseGuideL_Cyl_Var.In_AutoHome	:= FALSE;
			ER_CaseGuideR_Cyl_Var.In_AutoWork	:= TRUE;
			ER_CaseGuideR_Cyl_Var.In_AutoHome	:= FALSE;

			
			(*Wait for BFlap and Vacuum Switch to enable the CaseGuide*)
			IF ER_BFlapR_Cyl_Var.S_WorkPos AND 
				ER_BFlapL_Cyl_Var.S_WorkPos AND
				(((*ER_BFlapR_Vac_Var.S_Vacuum AND *)ER_BFlapL_Vac_Var.S_Vacuum) OR MC.DryRun) THEN
					ER_CaseGuideL_Cyl_Var.In_AutoWork	:= TRUE;
					ER_CaseGuideL_Cyl_Var.In_AutoHome	:= FALSE;
					ER_CaseGuideR_Cyl_Var.In_AutoWork	:= TRUE;
					ER_CaseGuideR_Cyl_Var.In_AutoHome	:= FALSE;
					ER_TFlapOpnL_Cyl_Var.In_AutoWork	:= TRUE;
					ER_TFlapOpnL_Cyl_Var.In_AutoHome	:= FALSE;
					ER_TFlapOpnR_Cyl_Var.In_AutoWork	:= TRUE;
					ER_TFlapOpnR_Cyl_Var.In_AutoHome	:= FALSE;
			END_IF
	
			IF NOT MC.DryRun THEN
				ER_BFlapR_Vac_Var.In_AutoVacuum := TRUE;
				ER_BFlapR_Vac_Var.In_AutoPurge := FALSE;
				ER_BFlapL_Vac_Var.In_AutoVacuum := TRUE;
				ER_BFlapL_Vac_Var.In_AutoPurge := FALSE;
			END_IF
			

			
			IF	ER_CaseGuideL_Cyl_Var.S_WorkPos AND
				ER_CaseGuideR_Cyl_Var.S_WorkPos THEN	
					ER_Arm_Vac_Var.In_AutoVacuum 	:= FALSE;
					ER_Arm_Vac_Var.In_AutoPurge 	:= TRUE;		
				
				IF ER_BFlapL_Cyl_Var.S_WorkPos AND 
					ER_BFlapR_Cyl_Var.S_WorkPos AND
					ER_TFlapOpnL_Cyl_Var.S_WorkPos AND
					ER_TFlapOpnR_Cyl_Var.S_WorkPos AND
					((ER_BFlapR_Vac_Var.S_Vacuum AND ER_BFlapL_Vac_Var.S_Vacuum) OR
					MC.DryRun)
					AND Station.Run_NextStepPls THEN
					ER_BFlapL_Cyl_Var.In_AutoWork := FALSE;
					ER_BFlapR_Cyl_Var.In_AutoWork := FALSE;
					ER_BFlapL_Vac_Var.In_AutoVacuum := FALSE;
					CaseBufferEmptying_Counter	:= CaseBufferEmptying_Counter + 1;
					GlueEmptying_Counter		:= GlueEmptying_Counter + 1;
					Station.RunStep := Station.RunStep + 10;
				END_IF
			END_IF	
	
	50 : 	(************* Bottom Flap Holder Cyl Down ****************)
			Station.Status 		:= '50: Bottom Flap Holder Cyl Down';
			Station.StatusInt	:= 256;
			ER_BFlapL_Cyl_Var.In_AutoWork := FALSE;
			ER_BFlapL_Cyl_Var.In_AutoHome := TRUE;
			ER_BFlapR_Cyl_Var.In_AutoWork := FALSE;
			ER_BFlapR_Cyl_Var.In_AutoHome := TRUE;
			
			IF ER_BFlapL_Cyl_Var.S_HomePos  
				AND ER_BFlapR_Cyl_Var.S_HomePos
				AND Station.Run_NextStepPls THEN
				ER_BFlapL_Cyl_Var.In_AutoHome := FALSE;
				ER_BFlapR_Cyl_Var.In_AutoHome := FALSE;
				Station.RunStep := Station.RunStep + 10;
			END_IF

	60 : 	(************* Rear and Front Side Moving Flap Close Cylinders Fwd ****************)
			Station.Status 		:= '60: Rear and Front Side Moving Flap Close Cylinders Fwd';
			Station.StatusInt	:= 257;
			
			IF Cfg_CollDircLtoR THEN
				ER_FFlapR_Cyl_Var.In_AutoWork := TRUE;
				ER_FFlapR_Cyl_Var.In_AutoHome := FALSE;
				ER_RFlapR_Cyl_Var.In_AutoWork := TRUE;
				ER_RFlapR_Cyl_Var.In_AutoHome := FALSE;			
			ELSE
				ER_FFlapL_Cyl_Var.In_AutoWork := TRUE;
				ER_FFlapL_Cyl_Var.In_AutoHome := FALSE;
				ER_RFlapL_Cyl_Var.In_AutoWork := TRUE;
				ER_RFlapL_Cyl_Var.In_AutoHome := FALSE;							
			END_IF
			
			IF (Cfg_CollDircLtoR AND 
				(ER_FFlapR_Cyl_Var.S_WorkPos AND ER_RFlapR_Cyl_Var.S_WorkPos)) OR
				(NOT Cfg_CollDircLtoR AND
				((ER_FFlapL_Cyl_Var.S_WorkPos AND ER_RFlapL_Cyl_Var.S_WorkPos))
				) AND Station.Run_NextStepPls THEN
				ER_FFlapR_Cyl_Var.In_AutoWork := FALSE;
				ER_RFlapR_Cyl_Var.In_AutoWork := FALSE;
				ER_FFlapL_Cyl_Var.In_AutoWork := FALSE;
				ER_RFlapL_Cyl_Var.In_AutoWork := FALSE;
				(*IF CO_YPush.Bypass THEN
					H_ER_CtnRdyForPushIn := FALSE;
					H_ER_CtnPushInDone := TRUE;
					H_ER_CtnSideFlapDone := FALSE;
				ELSE		*)			
					H_ER_CtnRdyForPushIn := TRUE;
					H_ER_CtnPushInDone := FALSE;
					H_ER_CtnSideFlapDone := FALSE;
				(*END_IF*)
				Station.RunStep := Station.RunStep + 10;
			END_IF
	
	70 : 	(************* Erector Arm Vacuum OFF ****************)
			Station.Status 		:= '70: Erector Arm Vacuum OFF';
			Station.StatusInt	:= 258;
			ER_Arm_Vac_Var.In_AutoVacuum := FALSE;
			ER_Arm_Vac_Var.In_AutoPurge := TRUE;

			(*IF ER_Arm_Vac_Var.S_Release THEN*)
				ER_Arm_Srv_Var.In_PosCmd := H_ER_Arm_Srv_CtnErectPos - 10;
				ER_Arm_Srv_Var.In_VelCmd := A_Srv_ErectorArmHiSpeed;
				ER_Arm_Srv_Var.In_MoveAbs := TRUE;
			(*END_IF*)
			
			IF ER_Arm_Vac_Var.S_Release AND 
				fcComparePos(CurrPos:= ER_Arm_Srv_Var.Out_CurrPos, TargetPos:= ER_Arm_Srv_Var.In_PosCmd,0.5) AND
				ER_Arm_Srv_Var.Out_InPos
				AND Station.Run_NextStepPls THEN
				ER_Arm_Vac_Var.In_AutoPurge := FALSE;
				ER_Arm_Srv_Var.In_MoveAbs := FALSE;
				Station.RunStep :=100;
			END_IF

	100 : 	(************* Erector Arm Cylinder Down ****************)
			(************* Right Top Open Home and Top Close Fwd ****************)
			Station.Status 		:= '75: Erector Arm Cylinder Down';
			Station.StatusInt	:= 259;
			ER_Arm_Cyl_Var.In_AutoHome 			:= FALSE;
			ER_Arm_Cyl_Var.In_AutoWork 			:= TRUE;
			
			
			IF NOT End_Production THEN
				
			IF Cfg_CollDircLtoR THEN
				ER_TFlapOpnR_Cyl_Var.In_AutoWork	:= FALSE;
				ER_TFlapOpnR_Cyl_Var.In_AutoHome	:= TRUE;
			(*
				ER_TFlapClsR_Cyl_Var.In_AutoWork	:= TRUE;
				ER_TFlapClsR_Cyl_Var.In_AutoHome	:= FALSE;
			*)
			ELSE
				ER_TFlapOpnL_Cyl_Var.In_AutoWork	:= FALSE;
				ER_TFlapOpnL_Cyl_Var.In_AutoHome	:= TRUE;
			(*
				ER_TFlapClsL_Cyl_Var.In_AutoWork	:= TRUE;
				ER_TFlapClsL_Cyl_Var.In_AutoHome	:= FALSE;
			*)
			END_IF
			END_IF
			
			IF ER_Arm_Cyl_Var.S_WorkPos
				AND Station.Run_NextStepPls THEN
				ER_Arm_Cyl_Var.In_AutoWork := FALSE;
				Station.RunStep := Station.RunStep + 10;
			END_IF

	110 : 	(************* Erector Arm Servo Move Back to Home Position ****************)
			Station.Status 		:= '80: Erector Arm Servo Move Back to Home Position';
			Station.StatusInt	:= 260;
			
			ER_Arm_Srv_Var.In_PosCmd := H_ER_Arm_Srv_CtnVacuumPos;
			ER_Arm_Srv_Var.In_VelCmd := A_Srv_ErectorArmHiSpeed;
			ER_Arm_Srv_Var.In_MoveAbs := TRUE;
			
			IF fcComparePos(CurrPos:= ER_Arm_Srv_Var.Out_CurrPos, TargetPos:= ER_Arm_Srv_Var.In_PosCmd,0.5) AND
				ER_Arm_Srv_Var.Out_InPos 
				AND Station.Run_NextStepPls THEN				
				ER_Arm_Srv_Var.In_MoveAbs := FALSE;
				Station.RunStep := Station.RunStep + 10;	
			END_IF
			
	120 : 	(************* Erector Arm Cylinder Up Then Tilt Fwd ****************)
			Station.Status 		:= '90: Erector Arm Cylinder Up and Tilt Fwd';
			Station.StatusInt	:= 261;
			
			ER_Arm_Cyl_Var.In_AutoWork := FALSE;
			ER_Arm_Cyl_Var.In_AutoHome := TRUE;
			
			IF ER_Arm_Cyl_Var.S_HomePos THEN
				ER_ArmTilt_Cyl_Var.In_AutoHome := FALSE;
				ER_ArmTilt_Cyl_Var.In_AutoWork := TRUE;
			END_IF	

			IF ER_Arm_Cyl_Var.S_HomePos AND ER_ArmTilt_Cyl_Var.S_WorkPos
				AND Station.Run_NextStepPls THEN	
				ER_Arm_Cyl_Var.In_AutoHome := FALSE;
				ER_ArmTilt_Cyl_Var.In_AutoWork := FALSE;
				Station.RunStep := 1000;						
			END_IF
		
	1000 : 	(************* Process Done ****************)
			Station.Status 		:= '1000: Process Done';
			Station.StatusInt	:= 499;
			
			M_StepRun := FALSE;
			Station.RunStep := 0;
			

	END_CASE


ELSE
	Station.RunStep := 0;
	
	IF Station.MajorFault OR Station.MinorFault THEN
		Station.Status 		:= 'Station Error';
		Station.StatusInt	:= 4;
	ELSIF Station.Origin THEN
		Station.Status 		:= 'Station In Origin';
		Station.StatusInt	:= 5;
	ELSIF NOT Station.OriginSchRun AND NOT MC.OriginSchRun THEN
		Station.Status 		:= 'Station Not In Origin';
		Station.StatusInt	:= 6;
	END_IF
END_IF

(*Station.Running := (Station.RunStep>0);*)

END_PROGRAM

// ---- POUs/Erector/ER_Auto_FixedFlap.TcPOU
PROGRAM ER_Auto_FixedFlap
VAR_IN_OUT
	Station		:structStationCtrl;
END_VAR
VAR
	Timeout	:TON;	
	StpCtnPE_TOFF: Ton;
END_VAR

(**************************************************************************************************************)
(* GENERAL STATION MAPPING  *)
(**************************************************************************************************************)
(*Station.Name			:=	'CARTON ERECTOR & SIDE FLAP CLOSING';*)
Station.Rdy 			:= 	Station.Origin;
Station.AutoRun 		:=	(MC.AutoRunning OR Station.M_Step) AND 
							NOT (Station.Bypass OR Station.MajorFault OR Station.MinorFault);
ER_FixedFlap.RunReq		:= 	(H_ER_CtnPushInDone AND NOT H_ER_CtnSideFlapDone)			
							(*OR MC.DryRun OR Station.M_Step*) ;
ER_FixedFlap.RunCond	:=	(NOT CO_YPush.Running OR 
							(	CO_YPush.RunStep>=120 AND 
								CO_FlapGuide_Cyl_Var.S_HomePos AND 
								CO_Brdg_Cyl_Var.S_HomePos AND 
								CO_YPush_Strk_Cyl_Var.S_HomePos)) AND (*Y Pusher not pushing stack forward*)
							(*NOT Station.Running AND	*)							(*Erector Arm Not Running*)
							NOT (Station.Done OR MC.StopPressed);
Station.Run_NextStepPls	:=	(Station.AutoRun AND NOT Station.M_Step) OR 
							(Station.M_Step AND M_StepFwdPls) OR HMI.T_OneCycleRun;
Station.Run_PrevStepPls	:=	(Station.M_Step AND M_StepBwdPls);

(**************************************************************************************************************)
(* Auto Sequance*)
(**************************************************************************************************************)

IF Station.AutoRun OR Station.M_Step THEN

	CASE ER_FixedFlap.RunStep OF

	0 : 	(************* Ready To Run ****************)
			IF ER_FixedFlap.RunCond AND ER_FixedFlap.RunReq THEN
				ER_FixedFlap.RunStep := ER_FixedFlap.RunStep + 10;	(*Activate Side Flap Closing*)
			END_IF

	10 : 	(************* Rear and Front Side Fixed Flap Close Cylinders Fwd ****************)
			Station.Status 		:= '10: Side Fixed Flap Close Cylinders Fwd';
			Station.StatusInt	:= 270;
			
			IF Cfg_CollDircLtoR THEN
				ER_FFlapL_Cyl_Var.In_AutoWork := TRUE;
				ER_FFlapL_Cyl_Var.In_AutoHome := FALSE;		
				IF ER_FFlapL_Cyl_Var.S_WorkPos THEN
					ER_RFlapL_Cyl_Var.In_AutoWork := TRUE;
					ER_RFlapL_Cyl_Var.In_AutoHome := FALSE;		
				END_IF	
			ELSE
				ER_FFlapR_Cyl_Var.In_AutoWork := TRUE;
				ER_FFlapR_Cyl_Var.In_AutoHome := FALSE;
				IF ER_FFlapR_Cyl_Var.S_WorkPos THEN
					ER_RFlapR_Cyl_Var.In_AutoWork := TRUE;
					ER_RFlapR_Cyl_Var.In_AutoHome := FALSE;		
				END_IF						
			END_IF
			
			IF (Cfg_CollDircLtoR AND 
				(ER_FFlapL_Cyl_Var.S_WorkPos AND ER_RFlapL_Cyl_Var.S_WorkPos)) OR
				(NOT Cfg_CollDircLtoR AND
				((ER_FFlapR_Cyl_Var.S_WorkPos AND ER_RFlapR_Cyl_Var.S_WorkPos))
				) AND Station.Run_NextStepPls THEN
				ER_FFlapR_Cyl_Var.In_AutoWork := FALSE;
				ER_RFlapR_Cyl_Var.In_AutoWork := FALSE;
				ER_FFlapL_Cyl_Var.In_AutoWork := FALSE;
				ER_RFlapL_Cyl_Var.In_AutoWork := FALSE;
				ER_FixedFlap.RunStep := ER_FixedFlap.RunStep + 10;
			END_IF
			
	20 : 	(************* Bottom Flap Holder Vacuum OFF ****************)
			Station.Status 		:= '20: Bottom Flap Holder Vacuum OFF';
			Station.StatusInt	:= 271;
			
			(*ER_BFlapR_Vac_Var.In_AutoVacuum := FALSE;
			ER_BFlapR_Vac_Var.In_AutoPurge := TRUE;*)
			ER_BFlapL_Vac_Var.In_AutoVacuum := FALSE;
			ER_BFlapL_Vac_Var.In_AutoPurge := TRUE;
			
			IF (*ER_BFlapR_Vac_Var.S_Release AND*) ER_BFlapL_Vac_Var.S_Release AND
				Station.Run_NextStepPls THEN
				ER_BFlapL_Cyl_Var.In_AutoWork := FALSE;
				ER_BFlapR_Cyl_Var.In_AutoWork := FALSE;
				(*ER_BFlapR_Vac_Var.In_AutoVacuum := FALSE;*)
				ER_BFlapL_Vac_Var.In_AutoVacuum := FALSE;
				ER_FixedFlap.RunStep := ER_FixedFlap.RunStep + 10;
			END_IF


	30 : 	(************* Bottom Flap Vacuum Off ****************)
			Station.Status := '30: Bottom Flap Close Vacuum Off';
			Station.StatusInt	:= 271;
			
				(*ER_BFlapR_Vac_Var.In_AutoVacuum := FALSE;
				ER_BFlapR_Vac_Var.In_AutoPurge := TRUE;*)
				ER_BFlapL_Vac_Var.In_AutoVacuum := FALSE;
				ER_BFlapL_Vac_Var.In_AutoPurge := TRUE;
			
			IF 	ER_BFlapL_Vac_Var.S_Release (*AND 
				ER_BFlapR_Vac_Var.S_Release*) AND 
				Station.Run_NextStepPls THEN
				ER_BFlapL_Cyl_Var.In_AutoWork := FALSE;
				ER_BFlapR_Cyl_Var.In_AutoWork := FALSE;
				ER_FixedFlap.RunStep := ER_FixedFlap.RunStep + 10;
			END_IF

			
	40 :	(************* Top Flap Close ****************)
			Station.Status 		:= '40: Top Flap Close';
			Station.StatusInt	:= 272;
			
			IF Cfg_CollDircLtoR THEN
					ER_TFlapClsL_Cyl_var.In_AutoWork 	:=TRUE;
					ER_TFlapClsL_Cyl_var.In_Autohome 	:=FALSE;
					ER_TFlapOpnL_Cyl_var.In_AutoWork 	:=FALSE;
					ER_TFlapOpnL_Cyl_var.In_Autohome 	:=TRUE;
					ER_TFlapClsR_Cyl_Var.In_AutoWork	:= TRUE;
					ER_TFlapClsR_Cyl_Var.In_AutoHome	:= FALSE;
					
				IF 	ER_TFlapClsL_Cyl_var.S_WorkPos  AND 
					ER_TFlapOpnL_Cyl_var.S_HomePos AND 
					Station.Run_NextStepPls THEN
					ER_TFlapClsL_Cyl_var.In_AutoWork 	:=FALSE;
					ER_TFlapOpnL_Cyl_var.In_Autohome 	:=FALSE;
					ER_FixedFlap.RunStep := ER_FixedFlap.RunStep + 10;
				END_IF
				
			ELSE
					ER_TFlapClsR_Cyl_var.In_AutoWork 	:=TRUE;
					ER_TFlapClsR_Cyl_var.In_Autohome 	:=FALSE;
					ER_TFlapOpnR_Cyl_var.In_AutoWork 	:=FALSE;
					ER_TFlapOpnR_Cyl_var.In_Autohome 	:=TRUE;
					ER_TFlapClsL_Cyl_Var.In_AutoWork	:= TRUE;
					ER_TFlapClsL_Cyl_Var.In_AutoHome	:= FALSE;
					
				IF 	ER_TFlapClsR_Cyl_var.S_WorkPos  AND 
					ER_TFlapOpnR_Cyl_var.S_HomePos AND 
					Station.Run_NextStepPls THEN
					ER_TFlapClsR_Cyl_var.In_AutoWork 	:=FALSE;
					ER_TFlapOpnR_Cyl_var.In_Autohome 	:=FALSE;
					ER_FixedFlap.RunStep := ER_FixedFlap.RunStep + 10;
				END_IF
				
			
			END_IF


	
	50 : 	(************* All Side Flap Close Cylinders Bwd ****************)
			Station.Status 		:= '50: All Side Flap Close Cylinders Bwd';
			Station.StatusInt	:= 273;
			
			ER_FFlapL_Cyl_Var.In_AutoWork := FALSE;
			ER_FFlapL_Cyl_Var.In_AutoHome := TRUE;
			ER_FFlapR_Cyl_Var.In_AutoWork := FALSE;
			ER_FFlapR_Cyl_Var.In_AutoHome := TRUE;
			
			IF ER_FFlapL_Cyl_Var.S_HomePos AND 
				ER_FFlapR_Cyl_Var.S_HomePos AND
				Station.Run_NextStepPls THEN
				ER_FFlapR_Cyl_Var.In_AutoHome := FALSE;
				ER_RFlapR_Cyl_Var.In_AutoHome := FALSE;
				ER_FFlapL_Cyl_Var.In_AutoHome := FALSE;
				ER_RFlapL_Cyl_Var.In_AutoHome := FALSE;
				ER_FixedFlap.RunStep := 1000;
			END_IF

	1000 : 	(************* Process Done ****************)
			Station.Status 			:= '1000: Process Done';
			Station.StatusInt		:= 499;
			M_StepRun := FALSE;
			H_ER_CtnSideFlapDone 	:= TRUE;
			H_ER_CtnPushInDone 		:= FALSE;
			H_ER_CtnRdyForPushIn 	:= FALSE;
			ER_FixedFlap.RunStep 	:= 0;
			

	END_CASE


ELSE
	
	ER_FixedFlap.RunStep := 0;
	
END_IF

Station.Running := (ER_FixedFlap.RunStep>0) OR (Station.RunStep>5);

END_PROGRAM

// ---- POUs/Erector/ER_Glue.TcPOU
PROGRAM ER_Glue
VAR_IN_OUT
	Station		:structStationCtrl;
END_VAR
VAR
	GlueStart1 				:BOOL;
	GlueStart2 				:BOOL;
	DistanceAdvanceForGlue	:REAL;
	CartonPreAtStopper		:BOOL;
	tmrNordsonNotRdy		:Ton;
	tmrNordsonOffDly		:Ton;
END_VAR

DistanceAdvanceForGlue	:=	(A_Srv_ErectorArmHiSpeed/60)*0.07;
				
H_ER_1St_GlueStartPos	:=	H_ER_ValveOffset + 
							CurrRecipe.rCaseA - 
							CurrRecipe.rGlue_Distance_Fr_Edge + DistanceAdvanceForGlue;

H_ER_1St_GlueStopPos	:=	H_ER_ValveOffset + 
							CurrRecipe.rCaseA - 
							CurrRecipe.rGlue_Distance_Fr_Edge -
							CurrRecipe.rGlue_Length + DistanceAdvanceForGlue;			

H_ER_2nd_GlueStartPos	:=	H_ER_ValveOffset + 
							CurrRecipe.rGlue_Distance_Fr_Edge + 
							CurrRecipe.rGlue_Length + DistanceAdvanceForGlue;

H_ER_2nd_GlueStopPos	:=	H_ER_ValveOffset + 
							CurrRecipe.rGlue_Distance_Fr_Edge +DistanceAdvanceForGlue;			

(**************** Glue Auto Sequence ****************************)
IF 	T_GlueEnable AND NOT mc.DryRun AND mc.AutoMode AND NOT tmrNordsonNotRdy.Q  THEN
	ER_Nordson_PumpOnOff_Var.In_AutoON	:=TRUE;
	ER_Nordson_HeaterOn_Var.In_AutoON	:=TRUE;
ELSE
	ER_Nordson_PumpOnOff_Var.In_AutoON	:=FALSE;
	ER_Nordson_HeaterOn_Var.In_AutoON	:=FALSE;
END_IF	

tmrNordsonNotRdy	(In:= NOT I_Nord_Rdy AND NOT tmrNordsonOffDly.Q, PT:= T#10S );
tmrNordsonOffDly	(In:= tmrNordsonNotRdy.Q, pt:= T#0.5S);


(********************* Glue Sequence Start ********************************)							
												
IF  (Station.RunStep  >= 0) AND
	(Station.RunStep  <= 20) AND
	I_ER_StpL_Ctn_PE AND
	I_ER_StpR_Ctn_PE THEN		
	CartonPreAtStopper	:=TRUE;

ELSIF Station.RunStep  >= 40 OR Station.RunStep  = 0	THEN
	CartonPreAtStopper	:=FALSE;
	
END_IF

GlueStart1	:= 	(ER_Arm_Srv_Var.Out_CurrPos 	<=	H_ER_1St_GlueStartPos )	AND				
				(ER_Arm_Srv_Var.Out_CurrPos 	>=	H_ER_1St_GlueStopPos );
GlueStart2	:= 	(ER_Arm_Srv_Var.Out_CurrPos 	<=	H_ER_2nd_GlueStartPos )	AND				
				(ER_Arm_Srv_Var.Out_CurrPos 	>=	H_ER_2nd_GlueStopPos );			
							
IF  (Station.RunStep  >= 20) AND
	(Station.RunStep <= 30)	AND		
	( GlueStart1 OR GlueStart2 ) AND
	CartonPreAtStopper AND
	T_GlueEnable	AND 
	(Station.AutoRun OR Station.M_Step) AND
	NOT mc.DryRun	THEN

ER_NordsonL_Cyl_var.In_AutoWork 	:=TRUE;
ER_NordsonL_Cyl_var.In_AutoHome 	:=FALSE;
ER_NordsonR_Cyl_var.In_AutoWork 	:=TRUE;
ER_NordsonR_Cyl_var.In_AutoHome 	:=FALSE;	

ELSE

ER_NordsonL_Cyl_var.In_AutoWork 	:=FALSE;
ER_NordsonL_Cyl_var.In_AutoHome 	:=TRUE;
ER_NordsonR_Cyl_var.In_AutoWork 	:=FALSE;
ER_NordsonR_Cyl_var.In_AutoHome 	:=TRUE;
	
END_IF								

(********************* Glue Sequence End ********************************)

END_PROGRAM

// ---- POUs/Erector/ER_Cylinder_Output.TcPOU
PROGRAM ER_Cylinder_Output
VAR
	bEnable:BOOL;
	Reset:BOOL;
	ER_TFlapOpnR_Cyl_Work_Tmr : TON;
END_VAR

bEnable := NOT MC.Trouble;

ER_FFlapL_Cyl_Var.In_HomeXLock := TRUE;
ER_FFlapL_Cyl_Var.In_WorkXLock := (NOT ER_Arm_Srv_Var.Out_Busy OR NOT ER_Arm_Vac_Var.S_Vacuum) (*AND
									(CO_YPush_Srv_Var.Out_CurrPos >= H_CO_YPush_Srv_CtnFinalPos+200)*);

ER_FFlapL_Cyl(				
	IN_CylName		:='FRONT FLAP CLOSE LEFT', 	
	In_Enable		:= bEnable, 	
	In_Reset		:= MC.ResetPressed, 	
	In_WorkRS		:= I_ER_FFlapL_Fwd, 	
	In_HomeRS		:= I_ER_FFlapL_Bwd, 	
	In_WorkTON		:= T#10MS, 	
	In_HomeTON		:= T#10MS, 	
	in_Timeout		:= TP_Cyl_Timeout, 	
	Out_WorkSV		=> O_ER_FFlapL_Fwd, 	
	Out_HomeSV		=> O_ER_FFlapL_Bwd, 	
	CylVar			:= ER_FFlapL_Cyl_Var,
	Station			:= SC[3]);

ER_BFlapL_Cyl_Var.In_HomeXLock := TRUE;
ER_BFlapL_Cyl_Var.In_WorkXLock := TRUE (*(NOT ER_Arm_Srv_Var.Out_Busy OR NOT ER_Arm_Vac_Var.S_Vacuum) AND
									(CO_YPush_Srv_Var.Out_CurrPos >= H_CO_YPush_Srv_CtnFinalPos+200) AND
									NOT CO_Brdg_Cyl_Var.S_WorkPos*) ;
		
ER_BFlapL_Cyl(				
	IN_CylName		:='BTM FLAP HOLD LEFT', 	
	In_Enable		:= bEnable, 	
	In_Reset		:= MC.ResetPressed, 	
	In_WorkRS		:= I_ER_BFlapL_Fwd, 	
	In_HomeRS		:= I_ER_BFlapL_Bwd, 	
	In_WorkTON		:= T#10MS, 	
	In_HomeTON		:= T#10MS, 	
	in_Timeout		:= TP_Cyl_Timeout, 	
	Out_WorkSV		=> O_ER_BFlapL_Fwd, 	
	Out_HomeSV		=> O_ER_BFlapL_Bwd, 	
	CylVar			:= ER_BFlapL_Cyl_Var,
	Station			:= SC[3]);

ER_StpL_Cyl_Var.In_HomeXLock := TRUE;
ER_StpL_Cyl_Var.In_WorkXLock := TRUE;
				
ER_StpL_Cyl(				
	IN_CylName		:='STOPPER LEFT', 	
	In_Enable		:= bEnable, 	
	In_Reset		:= MC.ResetPressed, 	
	In_WorkRS		:= I_ER_StpL_Up, 	
	In_HomeRS		:= I_ER_StpL_Dn, 	
	In_WorkTON		:= T#10MS, 	
	In_HomeTON		:= T#10MS, 	
	in_Timeout		:= TP_Cyl_Timeout, 	
	Out_WorkSV		=> O_ER_StpL_Up, 	
	Out_HomeSV		=> O_ER_StpL_Dn, 	
	CylVar			:= ER_StpL_Cyl_Var,
	Station			:= SC[3]);

ER_FFlapR_Cyl_Var.In_HomeXLock := TRUE;
ER_FFlapR_Cyl_Var.In_WorkXLock := (NOT ER_Arm_Srv_Var.Out_Busy OR NOT ER_Arm_Vac_Var.S_Vacuum);
				
ER_FFlapR_Cyl(				
	IN_CylName		:='FRONT FLAP CLOSE RIGHT', 	
	In_Enable		:= bEnable, 	
	In_Reset		:= MC.ResetPressed, 	
	In_WorkRS		:= I_ER_FFlapR_Fwd, 	
	In_HomeRS		:= I_ER_FFlapR_Bwd, 	
	In_WorkTON		:= T#10MS, 	
	In_HomeTON		:= T#10MS, 	
	in_Timeout		:= TP_Cyl_Timeout, 	
	Out_WorkSV		=> O_ER_FFlapR_Fwd, 	
	Out_HomeSV		=> O_ER_FFlapR_Bwd, 	
	CylVar			:= ER_FFlapR_Cyl_Var,
	Station			:= SC[3]);

ER_BFlapR_Cyl_Var.In_HomeXLock := TRUE;
ER_BFlapR_Cyl_Var.In_WorkXLock := TRUE (* (NOT ER_Arm_Srv_Var.Out_Busy OR NOT ER_Arm_Vac_Var.S_Vacuum)*);
				
ER_BFlapR_Cyl(				
	IN_CylName		:='BTM FLAP HOLD RIGHT', 	
	In_Enable		:= bEnable, 	
	In_Reset		:= MC.ResetPressed, 	
	In_WorkRS		:= I_ER_BFlapR_Fwd, 	
	In_HomeRS		:= I_ER_BFlapR_Bwd, 	
	In_WorkTON		:= T#10MS, 	
	In_HomeTON		:= T#10MS, 	
	in_Timeout		:= TP_Cyl_Timeout, 	
	Out_WorkSV		=> O_ER_BFlapR_Fwd, 	
	Out_HomeSV		=> O_ER_BFlapR_Bwd, 	
	CylVar			:= ER_BFlapR_Cyl_Var,
	Station			:= SC[3]);

ER_StpR_Cyl_Var.In_HomeXLock := TRUE;
ER_StpR_Cyl_Var.In_WorkXLock := TRUE;
				
ER_StpR_Cyl(				
	IN_CylName		:='STOPPER RIGHT', 	
	In_Enable		:= bEnable, 	
	In_Reset		:= MC.ResetPressed, 	
	In_WorkRS		:= I_ER_StpR_Up, 	
	In_HomeRS		:= I_ER_StpR_Dn, 	
	In_WorkTON		:= T#10MS, 	
	In_HomeTON		:= T#10MS, 	
	in_Timeout		:= TP_Cyl_Timeout, 	
	Out_WorkSV		=> O_ER_StpR_Up, 	
	Out_HomeSV		=> O_ER_StpR_Dn, 	
	CylVar			:= ER_StpR_Cyl_Var,
	Station			:= SC[3]);

ER_Arm_Cyl_Var.In_HomeXLock := TRUE;
ER_Arm_Cyl_Var.In_WorkXLock := TRUE;
				
ER_Arm_Cyl(				
	IN_CylName		:='ARM UP/DN', 	
	In_Enable		:= bEnable, 	
	In_Reset		:= MC.ResetPressed, 	
	In_WorkRS		:= I_ER_Arm_Dn, 	
	In_HomeRS		:= I_ER_Arm_Up, 	
	In_WorkTON		:= T#10MS, 	
	In_HomeTON		:= T#10MS, 	
	in_Timeout		:= TP_Cyl_Timeout, 	
	Out_WorkSV		=> O_ER_Arm_Dn, 	
	Out_HomeSV		=> O_ER_Arm_Up, 	
	CylVar			:= ER_Arm_Cyl_Var,
	Station			:= SC[3]);

ER_ArmTilt_Cyl_Var.In_HomeXLock := TRUE;
ER_ArmTilt_Cyl_Var.In_WorkXLock := TRUE;
				
ER_ArmTilt_Cyl(				
	IN_CylName		:='ARM TILT', 	
	In_Enable		:= bEnable, 	
	In_Reset		:= MC.ResetPressed, 	
	In_WorkRS		:= I_ER_ArmTilt_Bwd, 	
	In_HomeRS		:= I_ER_ArmTilt_Fwd, 	
	In_WorkTON		:= T#10MS, 	
	In_HomeTON		:= T#10MS, 	
	in_Timeout		:= TP_Cyl_Timeout, 	
	Out_WorkSV		=> O_ER_ArmTilt_Bwd, 	
	Out_HomeSV		=> O_ER_ArmTilt_Fwd, 	
	CylVar			:= ER_ArmTilt_Cyl_Var,
	Station			:= SC[3]);

ER_RFlapL_Cyl_Var.In_HomeXLock := TRUE;
ER_RFlapL_Cyl_Var.In_WorkXLock := NOT CO_Brdg_Cyl_Var.S_WorkPos (*AND
									(CO_YPush_Srv_Var.Out_CurrPos >= H_CO_YPush_Srv_CtnFinalPos+200)*);
				
ER_RFlapL_Cyl(				
	IN_CylName		:='REAR FLAP CLOSE LEFT', 	
	In_Enable		:= bEnable, 	
	In_Reset		:= MC.ResetPressed, 	
	In_WorkRS		:= I_ER_RFlapL_Fwd, 	
	In_HomeRS		:= I_ER_RFlapL_Bwd, 	
	In_WorkTON		:= T#10MS, 	
	In_HomeTON		:= T#10MS, 	
	in_Timeout		:= TP_Cyl_Timeout, 	
	Out_WorkSV		=> O_ER_RFlapL_Fwd, 	
	Out_HomeSV		=> O_ER_RFlapL_Bwd, 	
	CylVar			:= ER_RFlapL_Cyl_Var,
	Station			:= SC[3]);

ER_RFlapR_Cyl_Var.In_HomeXLock := TRUE;
ER_RFlapR_Cyl_Var.In_WorkXLock := TRUE;

ER_RFlapR_Cyl(				
	IN_CylName		:='REAR FLAP CLOSE RIGHT', 
	In_Enable		:= bEnable, 	
	In_Reset		:= MC.ResetPressed, 	
	In_WorkRS		:= I_ER_RFlapR_Fwd, 	
	In_HomeRS		:= I_ER_RFlapR_Bwd, 	
	In_WorkTON		:= T#100MS, 	
	In_HomeTON		:= T#10MS, 	
	in_Timeout		:= TP_Cyl_Timeout, 	
	Out_WorkSV		=> O_ER_RFlapR_Fwd, 	
	Out_HomeSV		=> O_ER_RFlapR_Bwd, 	
	CylVar			:= ER_RFlapR_Cyl_Var,
	Station			:= SC[3]);

ER_CaseGuideL_Cyl_Var.In_HomeXLock := TRUE;
ER_CaseGuideL_Cyl_Var.In_WorkXLock := TRUE;

ER_CaseGuideL_Cyl(				
	IN_CylName		:='CASE GUIDE LEFT', 
	In_Enable		:= bEnable, 	
	In_Reset		:= MC.ResetPressed, 	
	In_WorkRS		:= I_ER_CaseGuideL_Fwd, 	
	In_HomeRS		:= I_ER_CaseGuideL_Bwd, 	
	In_WorkTON		:= T#10MS, 	
	In_HomeTON		:= T#10MS, 	
	in_Timeout		:= TP_Cyl_Timeout, 	
	Out_WorkSV		=> O_ER_CaseGuideL_Fwd	, 	
	Out_HomeSV		=> O_ER_CaseGuideL_Bwd	, 	
	CylVar			:= ER_CaseGuideL_Cyl_Var,
	Station			:= SC[3]);	
	
ER_CaseGuideR_Cyl_Var.In_HomeXLock := TRUE;
ER_CaseGuideR_Cyl_Var.In_WorkXLock := TRUE;

ER_CaseGuideR_Cyl(				
	IN_CylName		:='CASE GUIDE RIGHT', 
	In_Enable		:= bEnable, 	
	In_Reset		:= MC.ResetPressed, 	
	In_WorkRS		:= I_ER_CaseGuideR_Fwd, 	
	In_HomeRS		:= I_ER_CaseGuideR_Bwd, 	
	In_WorkTON		:= T#10MS, 	
	In_HomeTON		:= T#10MS, 	
	in_Timeout		:= TP_Cyl_Timeout, 	
	Out_WorkSV		=> O_ER_CaseGuideR_Fwd	, 	
	Out_HomeSV		=> O_ER_CaseGuideR_Bwd	, 	
	CylVar			:= ER_CaseGuideR_Cyl_Var,
	Station			:= SC[3]);		
	

ER_TFlapOpnL_Cyl_Var.In_HomeXLock := TRUE;
ER_TFlapOpnL_Cyl_Var.In_WorkXLock := ER_TFlapClsL_Cyl_Var.S_HomePos;

ER_TFlapOpnL_Cyl(				
	IN_CylName		:='TOP FLAP OPN LEFT', 
	In_Enable		:= bEnable, 	
	In_Reset		:= MC.ResetPressed, 	
	In_WorkRS		:= I_ER_TFlapOpnL_Fwd, 	
	In_HomeRS		:= I_ER_TFlapOpnL_Bwd, 	
	In_WorkTON		:= T#10MS, 	
	In_HomeTON		:= T#10MS, 	
	in_Timeout		:= TP_Cyl_Timeout, 	
	Out_WorkSV		=> O_ER_TFlapOpnL_Fwd, 	
	Out_HomeSV		=> O_ER_TFlapOpnL_Bwd, 	
	CylVar			:= ER_TFlapOpnL_Cyl_Var,
	Station			:= SC[3]);	
				
ER_TFlapClsL_Cyl_Var.In_HomeXLock := TRUE;
ER_TFlapClsL_Cyl_Var.In_WorkXLock := ER_TFlapOpnL_Cyl_Var.S_HomePos;

ER_TFlapClsL_Cyl(				
	IN_CylName		:='TOP FLAP CLS LEFT', 
	In_Enable		:= bEnable, 	
	In_Reset		:= MC.ResetPressed, 	
	In_WorkRS		:= I_ER_TFlapClsL_Fwd, 	
	In_HomeRS		:= I_ER_TFlapClsL_Bwd, 	
	In_WorkTON		:= T#10MS, 	
	In_HomeTON		:= T#10MS, 	
	in_Timeout		:= TP_Cyl_Timeout, 	
	Out_WorkSV		=> O_ER_TFlapClsL_Fwd, 	
	Out_HomeSV		=> O_ER_TFlapClsL_Bwd, 	
	CylVar			:= ER_TFlapClsL_Cyl_Var,
	Station			:= SC[3]);
	
ER_TFlapOpnR_Cyl_Var.In_HomeXLock := TRUE;
ER_TFlapOpnR_Cyl_Var.In_WorkXLock := ER_TFlapClsR_Cyl_Var.S_HomePos;
ER_TFlapOpnR_Cyl_Work_Tmr(IN:= O_ER_TFlapOpnR_Fwd OR ER_TFlapOpnR_Cyl_Work_Tmr.Q AND NOT O_ER_TFlapOpnR_Bwd  ,PT:=T#0.7S);
ER_TFlapOpnR_Cyl(				
	IN_CylName		:='TOP FLAP OPN RIGHT', 
	In_Enable		:= bEnable, 	
	In_Reset		:= MC.ResetPressed, 	
	In_WorkRS		:= I_ER_TFlapOpnR_Fwd, 	
	In_HomeRS		:= I_ER_TFlapOpnR_Bwd, 	
	In_WorkTON		:= T#10MS, 	
	In_HomeTON		:= T#10MS, 	
	in_Timeout		:= TP_Cyl_Timeout, 	
	Out_WorkSV		=> O_ER_TFlapOpnR_Fwd, 	
	Out_HomeSV		=> O_ER_TFlapOpnR_Bwd, 	
	CylVar			:= ER_TFlapOpnR_Cyl_Var,
	Station			:= SC[3]);	
				
ER_TFlapClsR_Cyl_Var.In_HomeXLock := TRUE;
ER_TFlapClsR_Cyl_Var.In_WorkXLock := ER_TFlapOpnR_Cyl_Var.S_HomePos;

ER_TFlapClsR_Cyl(				
	IN_CylName		:='TOP FLAP CLS RIGHT', 
	In_Enable		:= bEnable, 	
	In_Reset		:= MC.ResetPressed, 	
	In_WorkRS		:= I_ER_TFlapClsR_Fwd, 	
	In_HomeRS		:= I_ER_TFlapClsR_Bwd, 	
	In_WorkTON		:= T#10MS, 	
	In_HomeTON		:= T#10MS, 	
	in_Timeout		:= TP_Cyl_Timeout, 	
	Out_WorkSV		=> O_ER_TFlapClsR_Fwd, 	
	Out_HomeSV		=> O_ER_TFlapClsR_Bwd, 	
	CylVar			:= ER_TFlapClsR_Cyl_Var,
	Station			:= SC[3]);
	
ER_NordsonL_Cyl_Var.In_HomeXLock := TRUE;
ER_NordsonL_Cyl_Var.In_WorkXLock := TRUE;

ER_NordsonL_Cyl(				
	IN_CylName		:='NORDSON LEFT VALVE', 
	In_Enable		:= bEnable, 	
	In_Reset		:= MC.ResetPressed, 	
	In_WorkRS		:= ER_NordsonL_Cyl.Out_WorkSV, 	
	In_HomeRS		:= ER_NordsonL_Cyl.Out_HomeSV, 	
	In_WorkTON		:= T#10MS, 	
	In_HomeTON		:= T#10MS, 	
	in_Timeout		:= TP_Cyl_Timeout, 	
	Out_WorkSV		=> O_Nord_ValveL_On, 	
	Out_HomeSV		=> , 	
	CylVar			:= ER_NordsonL_Cyl_Var,
	Station			:= SC[3]);	
	
ER_NordsonR_Cyl_Var.In_HomeXLock := TRUE;
ER_NordsonR_Cyl_Var.In_WorkXLock := TRUE;

ER_NordsonR_Cyl(				
	IN_CylName		:='NORDSON RIGHT VALVE', 
	In_Enable		:= bEnable, 	
	In_Reset		:= MC.ResetPressed, 	
	In_WorkRS		:= ER_NordsonR_Cyl.Out_WorkSV, 	
	In_HomeRS		:= ER_NordsonR_Cyl.Out_HomeSV, 	
	In_WorkTON		:= T#10MS, 	
	In_HomeTON		:= T#10MS, 	
	in_Timeout		:= TP_Cyl_Timeout, 	
	Out_WorkSV		=> O_Nord_ValveR_On, 	
	Out_HomeSV		=> , 	
	CylVar			:= ER_NordsonR_Cyl_Var,
	Station			:= SC[3]);

END_PROGRAM

// ---- POUs/Erector/ER_Servo_Output.TcPOU
PROGRAM ER_Servo_Output
VAR
	Reset:BOOL;
	bEnable:BOOL;
	plsStopMove: R_trig;
	debugcode: INT;
	debugcode2: INT;
END_VAR

IF (MC.AutoMode OR SC[3].M_Step) AND NOT ER.Bypass THEN
	ER_Arm_Srv_Var.In_ServoOn := TRUE;
	ER_WA_Srv_Var.In_ServoOn := FALSE;
END_IF

IF ER.OriginSchRun OR MC.OriginSchRun OR mc.AutoMode OR (mc.ResetPressed AND NOT mc.Trouble) THEN
	ER_Arm_Srv_Var.In_ServoOn := TRUE;
	ER_WA_Srv_Var.In_ServoOn := TRUE;
END_IF

(*plsStopMove(CLK:= NOT (SC[3].OriginSchRun OR MC.OriginSchRun OR SC[3].AutoRun));
IF plsStopMove.Q THEN
	ER_Arm_Srv_Var.In_StopMove := TRUE;
	ER_BufCvL_WA_Srv_Var.In_StopMove := TRUE;
	ER_FlapL_WA_Srv_Var.In_StopMove := TRUE;
	ER_BufCvR_WA_Srv_Var.In_StopMove := TRUE;
	ER_FlapR_WA_Srv_Var.In_StopMove := TRUE;
	ER_WA_Srv_Var.In_StopMove := TRUE;
END_IF*)

bEnable := NOT (SC[3].MajorFault or MC.Trouble);

ER_Arm_Srv_Var.In_MoveXLock := TRUE OR (*(CO_FFlapBrdg_Cyl_Var.S_HomePos AND
								CO_Brdg_Cyl_Var.S_HomePos AND
								CO_YPush_Srv_Var.Out_CurrPos <= H_CO_YPush_Srv_CtnFinalPos - 100) OR  debug*)
								SC[2].Bypass;

(*ER_Arm_Srv Erector Arm Motor - 10M1*)
ER_Arm_Srv_Drive(
	In_Enable:= bEnable AND NOT MC_WA_Run AND NOT Erector_SafetySensorBypass AND NOT E_Case_Infeed_Safety_NOk, 
	In_Reset := MC.ResetPressed,
	In_AbsEncoder:= TRUE, 
	In_DriveInput:= ER_Arm_Srv_Input, 
	In_CommState:= ER_Arm_Srv_State, 
	Out_DriveOutput=> ER_Arm_Srv_Output, 
	Out_DriveFeedRateOverride=> , 
	DriveVar:= ER_Arm_Srv_Var,
	Station			:= SC[3]);
IF (SC[3].MajorFault OR MC.Trouble)OR ER_Arm_Srv_State<>8 THEN
	debugcode := debugcode + 1;
END_IF
IF NOT ER_Arm_Srv_Drive.In_Enable THEN
	debugcode2 := debugcode2 + 1;
END_IF	
IF mc.ManualMode THEN	
	ER_Arm_Srv_Feedrate := 10000;
ELSE
	ER_Arm_Srv_Feedrate :=    INT_TO_UINT(hmi.V_MachineSpeed * 100);
END_IF


	
ER_WA_Srv_Var.In_MoveXLock := TRUE;
	
(*ER_WA_M5 Erector Width Adjust Motor 1 - 11M1*)
ER_WA_Srv_Drive(
	In_Enable:= bEnable, 
	In_Reset := MC.ResetPressed,
	In_AbsEncoder:= TRUE, 
	In_DriveInput:= ER_WA_Srv_Input, 
	In_CommState:= ER_WA_Srv_State, 
	Out_DriveOutput=> ER_WA_Srv_Output, 
	Out_DriveFeedRateOverride=> , 
	DriveVar:= ER_WA_Srv_Var,
	Station			:= SC[3]);


	IF mc.ManualMode THEN	
		ER_WA_Srv_Feedrate := 10000;
	ELSE
		ER_WA_Srv_Feedrate :=    INT_TO_UINT(hmi.V_MachineSpeed * 100);
	END_IF

END_PROGRAM

// ---- POUs/Erector/ER_Motor_Output.TcPOU
PROGRAM ER_Motor_Output
VAR
		bEnable:BOOL;
		Reset:BOOL;
END_VAR

bEnable := NOT MC.Trouble;

ER_BufCvL_Mtr_Var.In_MoveXLock := NOT  ER_BufCvL_Ctn_TON.Q;
	
ER_BufCvL_Mtr(
	IN_DevName:= 'CARTON BUFFER LEFT CV', 
	In_Enable:= bEnable, 
	In_Reset:= MC.ResetPressed, 
	In_StarterOK:= I_CartonCV_M1M2_OK, 
	Out_MotorOn=> O_ER_BufCv_Mtr1_On, 
	MotorVar:= ER_BufCvL_Mtr_Var,
	Station			:= SC[3]);

ER_BufCvR_Mtr_Var.In_MoveXLock := NOT  ER_BufCvR_Ctn_TON.Q;
	
ER_BufCvR_Mtr(
	IN_DevName:= 'CARTON BUFFER RIGHT CV', 
	In_Enable:= bEnable, 
	In_Reset:= MC.ResetPressed, 
	In_StarterOK:= I_CartonCV_M1M2_OK, 
	Out_MotorOn=> O_ER_BufCv_Mtr2_On, 
	MotorVar:= ER_BufCvR_Mtr_Var,
	Station			:= SC[3]);

END_PROGRAM

// ---- POUs/Erector/ER_Vacuum_Output.TcPOU
PROGRAM ER_Vacuum_Output
VAR
	bEnable: BOOL;
	Reset: BOOL;
END_VAR

bEnable := TRUE;

ER_BFlapL_Vac(
	IN_Name:= 'ERE. LEFT FLAP VACUUM', 
	In_Enable:= TRUE (*O_VacPump_On*), 
	In_Reset:= MC.ResetPressed, 
	In_Vacuum_Switch:= I_ER_BFlapL_VacSw, 
	In_Drop_Monitor_Enable:= FALSE, 
	In_VacuumTON:= T#200MS, 
	In_Release_TON:= T#0MS, 
	In_PurgeTON:= T#0MS, 
	in_Timeout:= T#15S,	(*debug*) 
	Out_VacuumSV=> o_ER_BFlapL_Vac_oN, 
	Out_PurgeSV=> , 
	VacVar:= ER_BFlapL_Vac_Var,
	Station			:= SC[3]);

ER_BFlapR_Vac_Var.In_AutoVacuum	:= 	ER_BFlapL_Vac_Var.In_AutoVacuum;
ER_BFlapR_Vac_Var.In_AutoPurge	:= 	ER_BFlapL_Vac_Var.In_AutoPurge;
ER_BFlapR_Vac_Var.In_OrgVacuum	:= 	ER_BFlapL_Vac_Var.In_OrgVacuum;
ER_BFlapR_Vac_Var.In_OrgPurge	:= 	ER_BFlapL_Vac_Var.In_OrgPurge;
ER_BFlapR_Vac_Var.T_ManVacuum	:= 	ER_BFlapL_Vac_Var.T_ManVacuum;
ER_BFlapR_Vac_Var.T_ManPurge	:= 	ER_BFlapL_Vac_Var.T_ManPurge;
	
ER_BFlapR_Vac(
	IN_Name:= 'ERE. RIGHT FLAP VACUUM', 
	In_Enable:= TRUE, 
	In_Reset:= MC.ResetPressed, 
	In_Vacuum_Switch:= I_ER_BFlapR_VacSw, 
	In_Drop_Monitor_Enable:= FALSE, 
	In_VacuumTON:= ER_BFlapL_Vac.In_VacuumTON, 
	In_Release_TON:= ER_BFlapL_Vac.In_Release_TON, 
	In_PurgeTON:= ER_BFlapL_Vac.In_PurgeTON, 
	in_Timeout:= ER_BFlapL_Vac.in_Timeout, 	
	Out_VacuumSV=> , 
	Out_PurgeSV=> , 
	VacVar:= ER_BFlapR_Vac_Var,
	Station			:= SC[3]);

	
ER_Arm_Vac(
	IN_Name:= 'ERE. ARM VACUUM', 
	In_Enable:= TRUE (*O_VacPump_On*), 
	In_Reset:= MC.ResetPressed, 
	In_Vacuum_Switch:= I_ER_Arm_VacSw, 
	In_Drop_Monitor_Enable:= NOT (SC[3].RunStep  >= 20 AND SC[3].RunStep <= 30) , 
	In_VacuumTON:= T#200MS, 
	In_Release_TON:= T#0MS, 
	In_PurgeTON:= T#0MS, 
	in_Timeout:= T#10S		(*debug*), 
	Out_VacuumSV=> o_ER_Arm_Vac_oN, 
	Out_PurgeSV=> , 
	VacVar:= ER_Arm_Vac_Var,
	Station			:= SC[3]);

END_PROGRAM

// ---- POUs/Exit/EX_Main.TcPOU
PROGRAM EX_Main
VAR
END_VAR

IF Cfg_BypassErector THEN
	HMI.T_Station_BypassP[4] := TRUE;
ELSE
	HMI.T_Station_BypassP[4] := FALSE;
END_IF

EX_Error	(Station:= SC[4]);
EX_Auto		(Station:= SC[4]);
EX_Origin	(Station:= SC[4]);

EX_Cylinder_Output();
EX_Servo_Output();
EX_Motor_Output();
EX_LoadCell_Output();

(* EX Structure is only for displaying on HMI*)
SC[4].T_OriginSearch := EX.T_OriginSearch;
EX := SC[4];

END_PROGRAM

// ---- POUs/Exit/EX_Error.TcPOU
PROGRAM EX_Error
VAR_IN_OUT
	Station		:structStationCtrl;
END_VAR

VAR
END_VAR

IF MC.ResetPressed THEN
	Station.SeqFaultWord := 0;
END_IF

(* 	Reserved Station.SeqFaultWord 
	= 1~49 for Major Fault
	= 100~149 for Origin Sequence Fault
	= 150~199 for Origin Width Adjust Sequence Fault
	= 200~299 for Auto Sequence Fault
	= 300~399 for misc fault listed on this page*)

Station.MajorFault := (Station.SeqFaultWord > 0) AND (Station.SeqFaultWord < 50);
Station.MinorFault := (Station.SeqFaultWord >= 100) OR 	Station.DeviceFault OR 
														E_WT_Conv_Jam OR 
														E_Weight_CV_CartonNotDetect or
														E_CartonTapingErrL OR 
														E_CartonTapingErrL;

END_PROGRAM

// ---- POUs/Exit/EX_Auto.TcPOU
PROGRAM EX_Auto
VAR_IN_OUT
	Station		:structStationCtrl;
END_VAR
VAR
	Timeout	:TON;	
	WT_Cv_CtnPE_TON: Ton;
	WT_Cv_DryRun: Ton;
	WT_Cyl_Hold: Ton;
	TimeoutTrigger: BOOL;
	TimeoutSetting: TIME;
END_VAR

(**************************************************************************************************************)
(* GENERAL STATION MAPPING  *)
(**************************************************************************************************************)
Station.Name			:=	'ERECTOR EXIT';
Station.Rdy 			:= 	Station.Origin;
Station.AutoRun 		:=	(MC.AutoRunning OR Station.M_Step OR (SC[5].M_Step AND SC[5].AutoRun)) AND 
							NOT (Station.Bypass OR Station.MajorFault OR Station.MinorFault);
Station.RunReq			:= 	((H_ER_CtnRdyForGlue OR I_EX_Cv_Ctn_PE) AND NOT H_ER_CtnGlueDone)
							OR (Station.M_Step AND NOT SC[5].M_Step);
Station.RunCond			:=	(NOT SC[3].Running OR SC[3].RunStep >= 40) AND	(*Erector Arm Not Running or finished pushing*)
							(NOT SC[5].Running OR SC[5].RunStep >= 70) AND	(*Elevator Not Running or Tilt Cylinders Back*)
							NOT (Station.Done OR (MC.StopPressed AND NOT (H_ER_CtnRdyForGlue AND NOT H_ER_CtnGlueDone))) AND
							NOT ((SC[5].M_Step AND SC[5].AutoRun));
Station.Run_NextStepPls	:=	(Station.AutoRun AND NOT Station.M_Step) OR 
							(Station.M_Step AND M_StepFwdPls) OR HMI.T_OneCycleRun;
Station.Run_PrevStepPls	:=	(Station.M_Step AND M_StepBwdPls);

(**************************************************************************************************************)
(* Auto Sequance*)
(**************************************************************************************************************)

Timeout(IN:=TimeoutTrigger, PT:=TimeoutSetting);
IF Timeout.Q THEN
	TimeoutTrigger := FALSE;
END_IF
WT_Cv_CtnPE_TON	(IN:= I_EX_Cv_Ctn_PE, PT:=T#0.1S);
WT_Cyl_Hold		(IN:= (EX_FlapHoldL_Cyl_Var.S_WorkPos AND EX_FlapHoldR_Cyl_Var.S_WorkPos), PT:=ER_GlueHold_Time * 1000);
WT_Cv_CtnPE_TON	(IN:= I_EX_Cv_Ctn_PE, PT:=T#100MS);
WT_Cv_DryRun	(IN:= WT_Mtr_Var.In_AutoON AND MC.DryRun, PT:=T#2S);
			
IF Station.AutoRun OR Station.M_Step THEN
	
	CASE Station.RunStep OF

	0 : 	(************* Ready To Run ****************)
			IF Station.RunCond AND Station.RunReq AND Station.Rdy THEN
				H_ER_CtnWeightOK 	:= FALSE;
				Station.RunStep 	:= Station.RunStep + 10;
			ELSIF NOT Station.RunCond THEN
				Station.Status 		:= '0: Station Waiting for Run Conditions';
				Station.StatusInt	:= 1;
			ELSIF NOT Station.RunReq THEN
				Station.Status 		:= '0: Station Waiting for Run Request';
				Station.StatusInt	:= 2;
			ELSE
				Station.Status 		:= '0: Station Not Ready';	
				Station.StatusInt	:= 3;			
			END_IF
			
		
	10 : 	(************* Run Conveyor Till Sensor Detects  ****************)
			Station.Status 		:= '10: Run Conveyor Till Sensor Detects Carton';
			Station.StatusInt	:= 301;
			(*
			Ex_SquarenessCylL_Var.In_AutoWork	:= FALSE;
			Ex_SquarenessCylL_Var.In_AutoHome 	:= TRUE; *)			
		(*
			IF T_GlueEnable THEN
				EX_StpCylL_Var.In_AutoHome	:=FALSE;
				EX_StpCylL_Var.In_Autowork	:=TRUE;
				EX_StpCylR_Var.In_AutoHome	:=FALSE;
				EX_StpCylR_Var.In_Autowork	:=TRUE;
			ELSE
				EX_StpCylL_Var.In_AutoHome	:=TRUE;
				EX_StpCylL_Var.In_Autowork	:=FALSE;
				EX_StpCylR_Var.In_AutoHome	:=TRUE;
				EX_StpCylR_Var.In_Autowork	:=false;	
			END_IF	*)
			
			EX_StpCylL_Var.In_AutoHome	:=FALSE;
			EX_StpCylL_Var.In_Autowork	:=TRUE;
			EX_StpCylR_Var.In_AutoHome	:=FALSE;
			EX_StpCylR_Var.In_Autowork	:=TRUE;
			
			WT_Mtr_Var.In_AutoON := TRUE;
			TimeoutTrigger := TRUE;
			TimeoutSetting := T#30S;
			
			
			
			WT_Cv_DryRun(IN:= WT_Mtr_Var.In_AutoON AND MC.DryRun, PT:=T#2S);
			
			IF WT_Cv_CtnPE_TON.Q  OR WT_Cv_DryRun.Q THEN
				TimeoutTrigger := FALSE;
				Station.RunStep := Station.RunStep + 10;
			ELSIF Timeout.Q THEN
				Station.SeqFaultWord 		:= 200;
				E_Weight_CV_CartonNotDetect	:= TRUE;
				Station.SeqFaultString 		:= 'Auto: Weight Conveyor Sensor Failed to detect Carton.';
			END_IF
			

	20 : 	(************* Flap Hold Cylinders Fwd  ****************)
			Station.Status 		:= '20: Flap Hold Cylinders Fwd';
			Station.StatusInt	:= 302;
(*						
IF NOT T_GlueEnable THEN
				EX_StpCylL_Var.In_AutoHome	:=TRUE;
				EX_StpCylL_Var.In_Autowork	:=FALSE;
				EX_StpCylR_Var.In_AutoHome	:=TRUE;
				EX_StpCylR_Var.In_Autowork	:=FALSE;
				WT_Mtr_Var.In_AutoON 		:= TRUE;
				Station.RunStep := Station.RunStep + 10;
				
			ELSE
				
					Ex_SquarenessCylL_Var.In_AutoWork	:= TRUE;
					Ex_SquarenessCylL_Var.In_AutoHome 	:= FALSE;	
					Ex_SquarenessCylR_Var.In_AutoWork	:= TRUE;
					Ex_SquarenessCylR_Var.In_AutoHome 	:= FALSE;	
	
					IF 	Ex_SquarenessCylL_Var.S_WorkPos AND 
						Ex_SquarenessCylL_Var.S_WorkPos  THEN
						EX_FlapHoldL_Cyl_Var.In_AutoWork 	:= TRUE;
						EX_FlapHoldL_Cyl_Var.In_AutoHome 	:= FALSE;
						EX_FlapHoldR_Cyl_Var.In_AutoWork 	:= TRUE;
						EX_FlapHoldR_Cyl_Var.In_AutoHome 	:= FALSE;
						WT_Mtr_Var.In_AutoON 				:= FALSE;
					END_IF
				
				
				IF ((WT_Cyl_Hold.Q AND
					EX_FlapHoldL_Cyl_Var.S_WorkPos AND
					EX_FlapHoldR_Cyl_Var.S_WorkPos AND
					Ex_SquarenessCylL_Var.S_WorkPos AND
					Ex_SquarenessCylR_Var.S_WorkPos ) OR
					NOT T_GlueEnable)	 AND
					Station.Run_NextStepPls THEN
					EX_FlapHoldL_Cyl_Var.In_AutoWork := FALSE;
					EX_FlapHoldR_Cyl_Var.In_AutoWork := FALSE;
					EX_StpCylL_Var.In_AutoHome	:=TRUE;
					EX_StpCylL_Var.In_Autowork	:=FALSE;
					EX_StpCylR_Var.In_AutoHome	:=TRUE;
					EX_StpCylR_Var.In_Autowork	:=FALSE;	
					Station.RunStep := Station.RunStep + 10;
				END_IF
			END_IF
*)		
				
					Ex_SquarenessCylL_Var.In_AutoWork	:= TRUE;
					Ex_SquarenessCylL_Var.In_AutoHome 	:= FALSE;	
					Ex_SquarenessCylR_Var.In_AutoWork	:= TRUE;
					Ex_SquarenessCylR_Var.In_AutoHome 	:= FALSE;	
	
					IF 	Ex_SquarenessCylL_Var.S_WorkPos AND 
						Ex_SquarenessCylL_Var.S_WorkPos  THEN
						EX_FlapHoldL_Cyl_Var.In_AutoWork 	:= TRUE;
						EX_FlapHoldL_Cyl_Var.In_AutoHome 	:= FALSE;
						EX_FlapHoldR_Cyl_Var.In_AutoWork 	:= TRUE;
						EX_FlapHoldR_Cyl_Var.In_AutoHome 	:= FALSE;
						WT_Mtr_Var.In_AutoON 				:= FALSE;
					END_IF
				
				
				IF ((WT_Cyl_Hold.Q AND
					EX_FlapHoldL_Cyl_Var.S_WorkPos AND
					EX_FlapHoldR_Cyl_Var.S_WorkPos AND
					Ex_SquarenessCylL_Var.S_WorkPos AND
					Ex_SquarenessCylR_Var.S_WorkPos ))AND
					Station.Run_NextStepPls THEN
					EX_FlapHoldL_Cyl_Var.In_AutoWork := FALSE;
					EX_FlapHoldR_Cyl_Var.In_AutoWork := FALSE;
					EX_StpCylL_Var.In_AutoHome	:=TRUE;
					EX_StpCylL_Var.In_Autowork	:=FALSE;
					EX_StpCylR_Var.In_AutoHome	:=TRUE;
					EX_StpCylR_Var.In_Autowork	:=FALSE;	
					Station.RunStep := Station.RunStep + 10;
				END_IF
	30 : 	(************* Flap Hold Cylinders Bwd ****************)
			Station.Status 		:= '30: Flap Hold Cylinders Bwd';
			Station.StatusInt	:= 303;
	

			EX_FlapHoldL_Cyl_Var.In_AutoWork 	:= FALSE;
			EX_FlapHoldL_Cyl_Var.In_AutoHome 	:= TRUE;
			EX_FlapHoldR_Cyl_Var.In_AutoWork 	:= FALSE;
			EX_FlapHoldR_Cyl_Var.In_AutoHome 	:= TRUE;
			
			
			
			Ex_SquarenessCylL_Var.In_AutoWork	:= FALSE;
			Ex_SquarenessCylL_Var.In_AutoHome 	:= TRUE;
			Ex_SquarenessCylR_Var.In_AutoWork	:= FALSE;
			Ex_SquarenessCylR_Var.In_AutoHome 	:= TRUE;
		
			EX_StpCylL_Var.In_AutoHome			:=TRUE;
			EX_StpCylL_Var.In_Autowork			:=FALSE;
			EX_StpCylR_Var.In_AutoHome			:=TRUE;
			EX_StpCylR_Var.In_Autowork			:=FALSE;
			WT_Mtr_Var.In_AutoON 				:= FALSE;(*
			H_ER_CtnGlueDone					:= true;*)
			
			IF 	EX_FlapHoldL_Cyl_Var.S_HomePos	AND
				EX_FlapHoldr_Cyl_Var.S_HomePos	AND
				Ex_SquarenessCylL_Var.S_HomePos AND
				Ex_SquarenessCylR_Var.S_HomePos AND
				EX_StpCylL_Var.S_HomePos AND
				EX_StpCylR_Var.S_HomePos AND
				Station.Run_NextStepPls THEN
					H_ER_CtnGlueDone 					:= TRUE;
					H_ER_CtnRdyForGlue 					:= FALSE;			
					EX_FlapHoldL_Cyl_Var.In_AutoHome 	:= FALSE;
					EX_FlapHoldR_Cyl_Var.In_AutoHome	:= FALSE;
					IF HOR.RunReq	AND (HOR.RunCond OR SC[6].Running)	 THEN
						Station.RunStep := 1000;
					END_IF	
			END_IF
	
	1000 : 	(************* Process Done ****************)
			Station.Status 		:= '1000: Process Done';
			Station.StatusInt	:= 499;
			
			M_StepRun := FALSE;
			Station.RunStep := 0;
			

	END_CASE


ELSE
	Station.RunStep := 0;
	
	IF Station.MajorFault OR Station.MinorFault THEN
		Station.Status 		:= 'Station Error';
		Station.StatusInt	:= 4;
	ELSIF Station.Origin THEN
		Station.Status 		:= 'Station In Origin';
		Station.StatusInt	:= 5;
	ELSIF NOT Station.OriginSchRun AND NOT MC.OriginSchRun THEN
		Station.Status 		:= 'Station Not In Origin';
		Station.StatusInt	:= 6;
	END_IF
END_IF

(*Station.Running := ((Station.RunStep>0) (*AND not (Station.RunStep =30 AND station.Origin *))  OR sc[6].Running;*)
Station.Running := Station.RunStep>0 OR (sc[6].RunStep>0 and sc[6].RunStep<20);

END_PROGRAM

// ---- POUs/Exit/EX_Origin.TcPOU
PROGRAM EX_Origin
VAR_IN_OUT
	Station		:structStationCtrl;
END_VAR
VAR
	EX_WA_Origin: BOOL;
	pls_OriginSchRun: R_trig;
	TimeoutTrigger: BOOL;
	TimeoutSetting: TIME;
	Timeout:ton;
	WidthAdjust_Tolerance	:REAL;
END_VAR

(**************************************************************************************************************)
(* Station Width Adjust in Origin Condition *)
(**************************************************************************************************************)
IF NOT MC_WA_Run THEN
	WidthAdjust_Tolerance	:=	5;
ELSE	
	WidthAdjust_Tolerance	:= 	1;
END_IF
	
EX_WA_Origin := 		(((fcComparePos(CurrPos:= EX_HeightL_WA_Srv_Var.Out_CurrPos, TargetPos:= H_EX_HeightL_WA_Srv_TargetPos, Tolerance := WidthAdjust_Tolerance)) AND
							NOT EX_HeightL_WA_Srv_Var.Out_Busy) AND
						((fcComparePos(CurrPos:= EX_HeightR_WA_Srv_Var.Out_CurrPos, TargetPos:= H_EX_HeightR_WA_Srv_TargetPos, Tolerance := WidthAdjust_Tolerance)) AND
							NOT EX_HeightR_WA_Srv_Var.Out_Busy)) ;

(**************************************************************************************************************)
(* Station Origin Condition *)
(**************************************************************************************************************)

Station.Origin 	:=	((EX_WA_Origin OR NOT MC_WA_Run )AND
					EX_FlapHoldL_Cyl_Var.S_HomePos AND
					EX_FlapHoldR_Cyl_Var.S_HomePos AND
					Ex_SquarenessCylL_Var.S_HomePos AND
					Ex_SquarenessCylR_Var.S_HomePos )	 OR
					Station.Bypass ;
					 		
(**************************************************************************************************************)
(* Station Origin Step *)
(**************************************************************************************************************)

pls_OriginSchRun(CLK:= MC.OriginSchRun OR Station.OriginSchRun);

Timeout(IN:=TimeoutTrigger, PT:=TimeoutSetting);
IF Timeout.Q THEN
	TimeoutTrigger := FALSE;
END_IF

IF (MC.OriginSchRun OR Station.OriginSchRun) AND NOT Station.Bypass   THEN
	CASE Station.OriginRunStep OF

	0 : 	(************* Ready To Run ****************)
			IF NOT Station.Origin AND pls_OriginSchRun.Q THEN
				Station.OriginRunStep := Station.OriginRunStep+10;	
			END_IF

	10 : 	(************* Flap Holder Cylinders Bwd ****************)
			(************* Stopper Up ****************)
			Station.Status 		:= 'Org10: Flap Holder Cylinders Bwd ';
			Station.StatusInt	:= 320;
			
			WT_Mtr_Var.In_OrgOn			:=FALSE;

			
			IF 	NOT EX_FlapHoldL_Cyl_Var.S_HomePos OR
				NOT EX_FlapHoldR_Cyl_Var.S_HomePos OR
				NOT Ex_SquarenessCylL_Var.S_HomePos OR
				NOT Ex_SquarenessCylR_Var.S_HomePos THEN
				EX_FlapHoldL_Cyl_Var.In_OrgHome := TRUE;
				EX_FlapHoldR_Cyl_Var.In_OrgHome := TRUE;
				Ex_SquarenessCylL_Var.In_OrgHome := TRUE;
				Ex_SquarenessCylR_Var.In_OrgHome := TRUE;
			ELSE
				EX_FlapHoldL_Cyl_Var.In_OrgHome := FALSE;
				EX_FlapHoldR_Cyl_Var.In_OrgHome := FALSE;
				Ex_SquarenessCylL_Var.In_OrgHome := FALSE;
				Ex_SquarenessCylR_Var.In_OrgHome := FALSE;
				
				Station.OriginRunStep := Station.OriginRunStep +10;
				

			END_IF
			
	20 : 	(************* Check Sensors Before Homing ****************)
			Station.Status 		:= 'Org20: Check Sensors Before Homing';
			Station.StatusInt	:= 321;
			
			IF (H_ER_CtnRdyForGlue OR H_ER_CtnGlueDone OR H_ER_CtnWeightOK) THEN
				WT_Mtr_Var.In_OrgOn := TRUE;
				TimeoutTrigger := TRUE;
				TimeoutSetting := T#5S;
			END_IF
			
			IF NOT WT_Mtr_Var.In_OrgOn OR Timeout.Q THEN
				WT_Mtr_Var.In_OrgOn := FALSE;
				IF (H_ER_CtnRdyForGlue OR H_ER_CtnGlueDone OR H_ER_CtnWeightOK)
					AND NOT I_EX_Cv_Ctn_PE THEN
					Station.SeqFaultWord 	:= 100;
					Station.SeqFaultString 	:= 'Origin: Carton Missing or Stuck on Erector Exit conveyor.';
					E_CartonMissing			:= TRUE;
				ELSIF NOT (H_ER_CtnRdyForGlue OR H_ER_CtnGlueDone OR H_ER_CtnWeightOK)
					AND I_EX_Cv_Ctn_PE THEN
					Station.SeqFaultWord 	:= 101;
					Station.SeqFaultString 	:= 'Origin: Carton Detected on Erector Exit is in undefined state. Remove Carton.';
					E_EX_CartonDetected		:= TRUE;
				END_IF
				
				IF  NOT MC_WA_Run  THEN
					Station.OriginRunStep := 0;
				ELSE
					Station.OriginRunStep := 1000;
				END_IF
			END_IF	
			
	

	1000 : 	(************* Check Sensor Before Width Adjust ****************)
			Station.Status 		:= 'Org1000: Check Sensor Before Width Adjust ';
			Station.StatusInt	:= 321;
			
			IF NOT EX_WA_Origin THEN
				IF I_EX_Cv_Ctn_PE THEN
					(* 150 - Carton Detected on Erector Exit conveyor. Remove Carton for Width Adjustment*)
					Station.SeqFaultWord := 150;
					Station.SeqFaultString := 'Origin: Carton Detected on Erector Exit conveyor. Remove Carton for Width Adjustment';
				ELSE
					Station.OriginRunStep := Station.OriginRunStep+10;		
				END_IF	
			ELSE
				Station.OriginRunStep := 0;	
			END_IF
			
	1010 : 	(************* Move Erector Exit and Height WA to the right width ****************)
			Station.Status 		:= 'Org1010: Move Erector Exit and Height WA to the right width ';
			Station.StatusInt	:= 322;
			(*
			EX_WA_Srv_Var.In_PosCmd := H_EX_WA_Srv_TargetPos;
			EX_WA_Srv_Var.In_VelCmd := A_Srv_WAOriginSpeed;
			(*Interlock movement to avoid collision with Erector WA*)
			IF H_EX_WA_Srv_TargetPos > EX_WA_Srv_Var.Out_CurrPos THEN	(*new width is bigger*)
				EX_WA_Srv_Var.In_MoveAbs := TRUE;
			ELSIF H_EX_WA_Srv_TargetPos < EX_WA_Srv_Var.Out_CurrPos AND 	(*new width is smaller*)
				EX_WA_Srv_Var.In_MoveXLock THEN
				EX_WA_Srv_Var.In_MoveAbs := TRUE;
			ELSE
				EX_WA_Srv_Var.In_MoveAbs := FALSE;
				EX_WA_Srv_Var.In_StopMove := TRUE;
			END_IF
			*)
			
			EX_HeightL_WA_Srv_Var.In_PosCmd := H_EX_HeightL_WA_Srv_TargetPos;
			EX_HeightL_WA_Srv_Var.In_VelCmd := A_Srv_WAOriginSpeed;
			EX_HeightL_WA_Srv_Var.In_MoveAbs := TRUE;

			EX_HeightR_WA_Srv_Var.In_PosCmd := H_EX_HeightR_WA_Srv_TargetPos;
			EX_HeightR_WA_Srv_Var.In_VelCmd := A_Srv_WAOriginSpeed;
			EX_HeightR_WA_Srv_Var.In_MoveAbs := TRUE;
			
			(*
			EX_TopL_WA_Srv_Var.In_PosCmd := H_EX_TopL_WA_Srv_TargetPos;
			EX_TopL_WA_Srv_Var.In_VelCmd := A_Srv_WAOriginSpeed;
			EX_TopL_WA_Srv_Var.In_MoveAbs := TRUE;

			EX_TopR_WA_Srv_Var.In_PosCmd := H_EX_TopR_WA_Srv_TargetPos;
			EX_TopR_WA_Srv_Var.In_VelCmd := A_Srv_WAOriginSpeed;
			EX_TopR_WA_Srv_Var.In_MoveAbs := TRUE;
			*)
			
			IF 	(fcComparePos(CurrPos:= EX_HeightL_WA_Srv_Var.Out_CurrPos, TargetPos:= EX_HeightL_WA_Srv_Var.In_PosCmd, Tolerance := 0.5) AND
						EX_HeightL_WA_Srv_Var.Out_InPos AND EX_HeightL_WA_Srv_Var.Out_Ready) AND
				(fcComparePos(CurrPos:= EX_HeightR_WA_Srv_Var.Out_CurrPos, TargetPos:= EX_HeightR_WA_Srv_Var.In_PosCmd, Tolerance := 0.5) AND
						EX_HeightR_WA_Srv_Var.Out_InPos AND EX_HeightR_WA_Srv_Var.Out_Ready) (*AND
				(fcComparePos(CurrPos:= EX_TopL_WA_Srv_Var.Out_CurrPos, TargetPos:= EX_TopL_WA_Srv_Var.In_PosCmd) AND
						EX_TopL_WA_Srv_Var.Out_InPos AND EX_TopL_WA_Srv_Var.Out_Ready) AND
				(fcComparePos(CurrPos:= EX_TopR_WA_Srv_Var.Out_CurrPos, TargetPos:= EX_TopR_WA_Srv_Var.In_PosCmd) AND
						EX_TopR_WA_Srv_Var.Out_InPos AND EX_TopR_WA_Srv_Var.Out_Ready)*) THEN

				EX_WA_Srv_Var.In_MoveAbs := FALSE;
				EX_HeightL_WA_Srv_Var.In_MoveAbs := FALSE;
				EX_HeightR_WA_Srv_Var.In_MoveAbs := FALSE;
				EX_TopL_WA_Srv_Var.In_MoveAbs := FALSE;
				EX_TopR_WA_Srv_Var.In_MoveAbs := FALSE;
				Station.OriginRunStep := 0;
			END_IF
						
	END_CASE

ELSE

	Station.OriginRunStep := 0;	
	TimeoutTrigger := FALSE;
	
END_IF

END_PROGRAM

// ---- POUs/Exit/EX_Cylinder_Output.TcPOU
PROGRAM EX_Cylinder_Output
VAR
	bEnableL: 	BOOL;
	bEnableR: 	BOOL;
	bEnable:	BOOL;
	Reset:	 	BOOL;
	TempStationStruct:structStationCtrl;
END_VAR

bEnableL := NOT MC.Trouble (*AND (NOT (SC[4].RunStep = 30) OR I_ER_FlapHoldL_Fwd)*);
bEnableR := NOT MC.Trouble (*AND (NOT (SC[4].RunStep = 30) OR I_ER_FlapHoldR_Fwd)*);
bEnable	 := NOT MC.Trouble;

EX_FlapHoldL_Cyl_Var.In_HomeXLock := TRUE;
EX_FlapHoldL_Cyl_Var.In_WorkXLock := TRUE;

EX_FlapHoldL_Cyl(				
	IN_CylName		:='(1Y8) FLAP HOLD', 	
	In_Enable		:= bEnableL, 	
	In_Reset		:= MC.ResetPressed, 	
	In_WorkRS		:= NOT I_ER_FlapHoldL_Bwd, 	
	In_HomeRS		:= I_ER_FlapHoldL_Bwd, 	
	In_WorkTON		:= T#500MS, 	
	In_HomeTON		:= T#100MS, 	
	in_Timeout		:= TP_Cyl_Timeout, 	
	Out_WorkSV		=> O_ER_FlapHoldL_Fwd, 	
	Out_HomeSV		=> O_ER_FlapHoldL_Bwd, 	
	CylVar			:= EX_FlapHoldL_Cyl_Var,
	Station			:= SC[4],
	Station2		:= SC[5]);

EX_FlapHoldR_Cyl_Var.In_HomeXLock := TRUE;
EX_FlapHoldR_Cyl_Var.In_WorkXLock := TRUE;

EX_FlapHoldR_Cyl(				
	IN_CylName		:='(2Y8) FLAP HOLD', 	
	In_Enable		:= bEnableR, 	
	In_Reset		:= MC.ResetPressed, 	
	In_WorkRS		:= NOT I_ER_FlapHoldR_Bwd, 	
	In_HomeRS		:= I_ER_FlapHoldR_Bwd, 	
	In_WorkTON		:= T#500MS, 	
	In_HomeTON		:= T#100MS, 	
	in_Timeout		:= TP_Cyl_Timeout, 	
	Out_WorkSV		=> O_EX_FlapHoldR_Fwd, 	
	Out_HomeSV		=> O_EX_FlapHoldR_Bwd, 	
	CylVar			:= EX_FlapHoldR_Cyl_Var,
	Station			:= SC[4],
	Station2		:= SC[5]);

EX_SquarenessCylL_Var.In_HomeXLock := TRUE;
EX_SquarenessCylL_Var.In_WorkXLock := TRUE;

EX_SquarenessCylL_Cyl(				
	IN_CylName		:='SQUARENESS CYL LEFT', 
	In_Enable		:= bEnable, 	
	In_Reset		:= MC.ResetPressed, 	
	In_WorkRS		:= I_EX_SquarenessL_Fwd, 	
	In_HomeRS		:= I_EX_SquarenessL_Bwd, 	
	In_WorkTON		:= T#100MS, 	
	In_HomeTON		:= T#10MS, 	
	in_Timeout		:= TP_Cyl_Timeout, 	
	Out_WorkSV		=> O_EX_SquarenessCylL_Fwd, 	
	Out_HomeSV		=> O_EX_SquarenessCylL_Bwd, 	
	CylVar			:= Ex_SquarenessCylL_Var,
	Station			:= SC[4]);

EX_SquarenessCylR_Var.In_HomeXLock := TRUE;
EX_SquarenessCylR_Var.In_WorkXLock := TRUE;

EX_SquarenessCylR_Cyl(				
	IN_CylName		:='SQUARENESS CYL RIGHT', 
	In_Enable		:= bEnable, 	
	In_Reset		:= MC.ResetPressed, 	
	In_WorkRS		:= I_EX_SquarenessR_Fwd, 	
	In_HomeRS		:= I_EX_SquarenessR_Bwd, 	
	In_WorkTON		:= T#100MS, 	
	In_HomeTON		:= T#10MS, 	
	in_Timeout		:= TP_Cyl_Timeout, 	
	Out_WorkSV		=> O_EX_SquarenessCylR_Fwd, 	
	Out_HomeSV		=> O_EX_SquarenessCylR_Bwd, 	
	CylVar			:= Ex_SquarenessCylR_Var,
	Station			:= SC[4]);				
				
EX_StpCylL_Var.In_HomeXLock := TRUE;
EX_StpCylL_Var.In_WorkXLock := TRUE;

EX_StpCylL_Cyl(				
	IN_CylName		:='EXIT STOPPER CYL LEFT', 
	In_Enable		:= bEnable, 	
	In_Reset		:= MC.ResetPressed, 	
	In_WorkRS		:= NOT I_EX_StpL_Dn, 	
	In_HomeRS		:= I_EX_StpL_Dn, 	
	In_WorkTON		:= T#100MS, 	
	In_HomeTON		:= T#10MS, 	
	in_Timeout		:= TP_Cyl_Timeout, 	
	Out_WorkSV		=> O_EX_StpCylL_Up, 	
	Out_HomeSV		=> O_EX_StpCylL_Dn, 	
	CylVar			:= EX_StpCylL_Var,
	Station			:= SC[4]);

EX_StpCylR_Var.In_HomeXLock := TRUE;
EX_StpCylR_Var.In_WorkXLock := TRUE;

EX_StpCylR_Cyl(				
	IN_CylName		:='EXIT STOPPER CYL RIGHT', 
	In_Enable		:= bEnable, 	
	In_Reset		:= MC.ResetPressed, 	
	In_WorkRS		:= NOT I_EX_StpR_Dn, 	
	In_HomeRS		:= I_EX_StpR_Dn, 	
	In_WorkTON		:= T#100MS, 	
	In_HomeTON		:= T#10MS, 	
	in_Timeout		:= TP_Cyl_Timeout, 	
	Out_WorkSV		=> O_EX_StpCylR_Up, 	
	Out_HomeSV		=> O_EX_StpCylR_Dn, 	
	CylVar			:= EX_StpCylR_Var,
	Station			:= SC[4]);

END_PROGRAM

// ---- POUs/Exit/EX_Servo_Output.TcPOU
PROGRAM EX_Servo_Output
VAR
	Reset:BOOL;
	EL_M2_Drive: INT;
	plsStopMove: R_trig;
	bEnable: BOOL;
END_VAR

IF (MC.AutoMode OR SC[4].M_Step) AND NOT EX.Bypass THEN
	EX_HeightL_WA_Srv_Var.In_ServoOn := FALSE;
	EX_HeightR_WA_Srv_Var.In_ServoOn := FALSE;
	EX_TopL_WA_Srv_Var.In_ServoOn := FALSE;
	EX_TopR_WA_Srv_Var.In_ServoOn := FALSE;
	EX_WA_Srv_Var.In_ServoOn := FALSE;
END_IF

IF EX.OriginSchRun OR MC.OriginSchRun THEN
	EX_HeightL_WA_Srv_Var.In_ServoOn := TRUE;
	EX_HeightR_WA_Srv_Var.In_ServoOn := TRUE;
	EX_TopL_WA_Srv_Var.In_ServoOn := TRUE;
	EX_TopR_WA_Srv_Var.In_ServoOn := TRUE;
	EX_WA_Srv_Var.In_ServoOn := TRUE;
END_IF

(*plsStopMove(CLK:= NOT (SC[4].OriginSchRun OR MC.OriginSchRun OR SC[4].AutoRun));
IF plsStopMove.Q THEN
	EX_HeightL_WA_Srv_Var.In_StopMove := TRUE;
	EX_HeightR_WA_Srv_Var.In_StopMove := TRUE;
	EX_TopL_WA_Srv_Var.In_StopMove := TRUE;
	EX_TopR_WA_Srv_Var.In_StopMove := TRUE;
	EX_WA_Srv_Var.In_StopMove := TRUE;
END_IF*)

bEnable := NOT (SC[4].MajorFault OR SC[4].MinorFault OR SC[4].DeviceFault OR MC.Trouble);

EX_HeightL_WA_Srv_Var.In_MoveXLock := EX_FlapHoldL_Cyl_Var.S_HomePos;

(*EX_WA_M1 Exit Left Height Width Adjust Motor - 112M1*)
EX_HeightL_WA_Srv_Drive(
	In_Enable:= TRUE (*Cfg_EnbAutoWA AND bEnable*), 
	In_Reset := MC.ResetPressed,
	In_AbsEncoder:= TRUE, 
	In_DriveInput:= EX_HeightL_WA_Srv_Input, 
	In_CommState:= EX_HeightL_WA_Srv_State, 
	Out_DriveOutput=> EX_HeightL_WA_Srv_Output, 
	Out_DriveFeedRateOverride=> (*EX_HeightL_WA_Srv_Feedrate*), 
	DriveVar:= EX_HeightL_WA_Srv_Var,
	Station			:= SC[4]);

	IF mc.ManualMode THEN	
		EX_HeightL_WA_Srv_Feedrate := 10000;
	ELSE
		EX_HeightL_WA_Srv_Feedrate :=    INT_TO_UINT(hmi.V_MachineSpeed * 100);
	END_IF
	
EX_HeightR_WA_Srv_Var.In_MoveXLock := EX_FlapHoldR_Cyl_Var.S_HomePos;
	
(*EX_WA_M2 Exit Right Height Width Adjust Motor - 113M1*)
EX_HeightR_WA_Srv_Drive(
	In_Enable:= TRUE(*Cfg_EnbAutoWA AND bEnable*), 
	In_Reset := MC.ResetPressed,
	In_AbsEncoder:= TRUE, 
	In_DriveInput:= EX_HeightR_WA_Srv_Input, 
	In_CommState:= 8(*EX_HeightR_WA_Srv_State*), 
	Out_DriveOutput=> EX_HeightR_WA_Srv_Output, 
	Out_DriveFeedRateOverride=> (*EX_HeightR_WA_Srv_Feedrate*), 
	DriveVar:= EX_HeightR_WA_Srv_Var,
	Station			:= SC[4]);
	
	IF mc.ManualMode THEN	
		EX_HeightR_WA_Srv_Feedrate := 10000;
	ELSE
		EX_HeightR_WA_Srv_Feedrate :=    INT_TO_UINT(hmi.V_MachineSpeed * 100);
	END_IF
(*
EX_TopL_WA_Srv_Var.In_MoveXLock := EX_FlapHoldL_Cyl_Var.S_HomePos;
	
(*EX_WA_M3 Exit Left Top Guide Adjust Motor - 124M1*)
EX_TopL_WA_Srv_Drive(
	In_Enable:= Cfg_EnbAutoWA AND bEnable, 
	In_Reset := MC.ResetPressed,
	In_AbsEncoder:= TRUE, 
	In_DriveInput:= EX_TopL_WA_Srv_Input, 
	In_CommState:= EX_TopL_WA_Srv_State, 
	Out_DriveOutput=> EX_TopL_WA_Srv_Output, 
	Out_DriveFeedRateOverride=> EX_TopL_WA_Srv_Feedrate, 
	DriveVar:= EX_TopL_WA_Srv_Var,
	Station			:= SC[4]);

EX_TopR_WA_Srv_Var.In_MoveXLock := EX_FlapHoldR_Cyl_Var.S_HomePos;

(*EX_WA_M5 Exit Right Top Guide Adjust Motor - 125M1*)
EX_TopR_WA_Srv_Drive(
	In_Enable:= Cfg_EnbAutoWA AND bEnable, 
	In_Reset := MC.ResetPressed,
	In_AbsEncoder:= TRUE, 
	In_DriveInput:= EX_TopR_WA_Srv_Input, 
	In_CommState:= EX_TopR_WA_Srv_State, 
	Out_DriveOutput=> EX_TopR_WA_Srv_Output, 
	Out_DriveFeedRateOverride=> EX_TopR_WA_Srv_Feedrate, 
	DriveVar:= EX_TopR_WA_Srv_Var,
	Station			:= SC[4]);

EX_WA_Srv_Var.In_MoveXLock := NOT I_EX_Cv_Ctn_PE AND 
								((EX_WA_Srv_Var.Out_CurrPos >= (ER_WA_Srv_Var.Out_CurrPos-20)) OR
								EX_WA_Srv_Var.Out_PosDirc);
	
(*EX_WA_M4 Erector Exit Width Adjust Motor - 114M1*)
EX_WA_Srv_Drive(
	In_Enable:= Cfg_EnbAutoWA AND bEnable AND FALSE (*debug due to mechanical*), 
	In_Reset := MC.ResetPressed,
	In_AbsEncoder:= TRUE, 
	In_DriveInput:= EX_WA_Srv_Input, 
	In_CommState:= EX_WA_Srv_State, 
	Out_DriveOutput=> EX_WA_Srv_Output, 
	
	Out_DriveFeedRateOverride=> EX_WA_Srv_Feedrate, 
	DriveVar:= EX_WA_Srv_Var,
	Station			:= SC[4]);
*)

END_PROGRAM

// ---- POUs/Exit/EX_Motor_Output.TcPOU
PROGRAM EX_Motor_Output
VAR
	Reset:BOOL;
	bEnable: BOOL;
	tmrWTCvMtr	:ton;
	
END_VAR

(******************** Error Stop ***********************)
IF E_WT_Conv_Jam THEN
	WT_Mtr_Var.E_OnErr	:= TRUE;
END_IF
(********************************************************)

bEnable := NOT MC.Trouble;

WT_Mtr_Var.In_MoveXLock := TRUE;

WT_Mtr(
	IN_DevName:= 'WEIGHT CHECKING CV', 
	In_Enable:= bEnable, 
	In_Reset:= MC.ResetPressed, 
	In_StarterOK:= I_Weighing_CV_OK, 
	Out_MotorOn=> O_Weighing_CV_ON, 
	MotorVar:= WT_Mtr_Var,
	Station			:= SC[4]);
	
	
tmrWTCvMtr(In:= O_Weighing_CV_ON AND (I_HOR_Entry_Cv_Present OR I_EX_Cv_Ctn_PE), PT:=T#30S);
E_WT_Conv_Jam := tmrWTCvMtr.Q;

END_PROGRAM

// ---- POUs/Exit/EX_LoadCell_Output.TcPOU
PROGRAM EX_LoadCell_Output
VAR

	plsInitVar: R_trig;
END_VAR

(*(*
	The SerialLineControl function block is supposed to be called in every PLC cycle.
	It communicates with the serial line hardware device and transmits or receives data.
	The SerialLineControl can be called in the standard task or in a separate fast task as well.
	A fast separate task will be necessary at high baud rates or 
	with KL6001 terminals which have a small process image (3 or 5 data bytes only)
*)

(*plsInitVar(CLK:=MC_Ctrl.In_EmgOK);*)
(*EX_LoadCellVar.In_Init := plsInitVar.Q;**)

EX_LoadCell(
	In_Enable:= Cfg_EnbWeightCheck, 
	In_Reset:= MC.ResetPressed, 
	Out_Trigger=> O_EX_HBM_Trigger, 
	TxBuffer:= TxBufferEL, 
	RxBuffer:= RxBufferEL, 
	HBM_Var:= EX_LoadCellVar,
	Station:=SC[4]);

*)

END_PROGRAM

// ---- POUs/Horizontal/HOR_Main.TcPOU
PROGRAM HOR_Main
VAR
	plsTestSequence: R_trig;
	TestSequencePos1: REAL;
	TestSequencePos2: REAL;
	TestSequenceInPos: Ton;
	TestSequenceStep: INT;
	HOR_LC_MuteTON: Ton;
	testbit: BOOL;
	MutingStartRtig	:R_TRIG;
END_VAR

IF Cfg_BypassHorizontal THEN
	HMI.T_Station_BypassP[6] := TRUE;
ELSE
	HMI.T_Station_BypassP[6] := FALSE;  
END_IF

HOR_Timers();

HOR_Error	(Station:= SC[6]);
HOR_Auto	(Station:= SC[6]);
HOR_Origin	(Station:= SC[6]);
Option_90Deg_Conv();
HOR_Servo_Output();
HOR_Motor_Output();

MutingStartRtig(CLK:= HOR_Tilt_Out_Mtr_Var.S_Running AND I_HOR_Tilt_In_Cv_Present , Q=> );
IF MutingStartRtig.Q THEN
	A_HOR_LC_Muting := TRUE;
END_IF	
IF HOR_LC_MuteTON.Q THEN
	A_HOR_LC_Muting := FALSE;
END_IF

HOR_LC_Muting 	:= A_HOR_LC_Muting;
HOR_LC_MuteTON 	(IN := O_HOR_LC_Mute1, pt := T#5S);
O_HOR_LC_Mute1 	:= HOR_LC_Muting;

(* HOR Structure is only for displaying on HMI*)
SC[6].T_OriginSearch := HOR.T_OriginSearch;
HOR := SC[6];

END_PROGRAM

// ---- POUs/Horizontal/HOR_Timers.TcPOU
PROGRAM HOR_Timers
VAR
END_VAR

HOR_Ctn_TON (IN := I_HOR_Entry_Cv_Present, pt := T#500MS);

HOR_Ctn_TOFF (IN := NOT I_HOR_Entry_Cv_Present , pt := T#500MS);

HOR_DnStream_TOFF (IN := NOT I_HOR_DnStream_Cv_Full, pt := T#500MS);


(*
HOR_TopCv_Ctn_TON (IN := I_EX_TopCV_Ctn_PE, pt := T#500MS);

HOR_TopCv_Ctn_TOFF (IN := NOT I_EX_TopCV_Ctn_PE, pt := T#1S);

HOR_BotCv_Ctn_TON (IN := I_EX_BotCV_Ctn_PE, pt := T#500MS);

HOR_BotCv_Ctn_TOFF (IN := NOT I_EX_BotCV_Ctn_PE, pt := T#3S);
*)

HOR_LC_Safety_TON (IN:= I_HLC_SC_OK, pt := T#100MS);

END_PROGRAM

// ---- POUs/Horizontal/HOR_Error.TcPOU
PROGRAM HOR_Error
VAR_IN_OUT
	Station		:structStationCtrl;
END_VAR

VAR
	Right_Tape_Err_NoReset	:BOOL;
	Left_Tape_Err_NoReset	:BOOL;	
	tmrTopCvMtr	:ton;
	tmrBtmCvMtr	:ton;

END_VAR

IF MC.ResetPressed THEN
	Station.SeqFaultWord := 0;
END_IF

(* 	Reserved Station.SeqFaultWord 
	= 1~49 for Major Fault
	= 100~149 for Origin Sequence Fault
	= 150~199 for Origin Width Adjust Sequence Fault
	= 200~299 for Auto Sequence Fault
	= 300~399 for misc fault listed on this page*)

Station.MajorFault := ((Station.SeqFaultWord > 0) AND (Station.SeqFaultWord < 50));
Station.MinorFault := (Station.SeqFaultWord >= 100) OR Station.DeviceFault
													OR E_Top_Conv_Jam 
													OR E_Bottom_Conv_Jam
													OR E_Weight_CV_CartonNotDetect 
													OR E_Hor_Entry_Sensor
													OR E_Hor_Exit_Sensor
													OR ((E_CartonTapingErrL 
													OR E_CartonTapingErrR 
													OR W_HOR_TapeLRefill 
													OR W_HOR_TapeRRefill
													OR E_Weigh_ConsecutiveErr) AND 
													NOT station.Running) ;

(* Tape Low Warning *)
IF WORD_TO_INT(HOR_Auto.CntTapeReal_SlotL.CV) >= TapeLow_Setting THEN
	W_Hor_TapeLowL	:= TRUE;
END_IF													
IF WORD_TO_INT(HOR_Auto.CntTapeReal_SlotR.CV) >= TapeLow_Setting THEN
	W_Hor_TapeLowR	:= TRUE;
END_IF	
IF E_Horizontal_LeftDoor_Opn THEN
	W_Hor_TapeLowL	:= FALSE;
END_IF
IF E_Horizontal_RightDoor_Opn THEN
	W_Hor_TapeLowR	:= FALSE;
END_IF


(*Tape Refill Warning*)					
W_HOR_TapeLRefill	:= MC.AutoMode AND NOT  Station.Bypass AND 
						NOT I_HOR_TapeL_Present_PE;
W_HOR_TapeRRefill	:= MC.AutoMode AND NOT  Station.Bypass AND 
						NOT I_HOR_TapeR_Present_PE;

(* Tape Error Reset *)						
IF E_Horizontal_RightDoor_Opn THEN 
	Right_Tape_Err_NoReset	:= TRUE;
END_IF
IF E_Horizontal_LeftDoor_Opn THEN 
	Left_Tape_Err_NoReset	:= TRUE;
END_IF

IF Right_Tape_Err_NoReset AND MC.ResetPressed THEN
	E_CartonTapingErrR		:=FALSE;
	Right_Tape_Err_NoReset	:= FALSE;
END_IF
IF Left_Tape_Err_NoReset AND MC.ResetPressed THEN
	E_CartonTapingErrL		:=FALSE;
	Left_Tape_Err_NoReset	:=FALSE;
END_IF

(* Weighing Error *)
IF Hor_Auto.Weight_Fail_Counter >= 3 and Cfg_EnbWeightCheck THEN
	E_Weigh_ConsecutiveErr := TRUE;
END_IF

(* Conveyor Jam Error *)
tmrTopCvMtr(In:= O_HOR_TopCv_Mtr_Run AND (I_HOR_Entry_Cv_Present OR I_EX_Cv_Ctn_PE), PT:=T#30S);
E_Top_Conv_Jam := tmrTopCvMtr.Q;

tmrBtmCvMtr(In:= O_HOR_BotCv_Mtr_Run AND (I_HOR_Entry_Cv_Present OR I_EX_Cv_Ctn_PE), PT:=T#30S);
E_Bottom_Conv_Jam :=tmrBtmCvMtr.Q;

END_PROGRAM

// ---- POUs/Horizontal/HOR_Auto.TcPOU
PROGRAM HOR_Auto
VAR_IN_OUT
	Station			:structStationCtrl;
END_VAR
VAR
	Timeout							:TON;	
	WT_Cv_CtnPE_TON					:Ton;
	ExitCvFull_TON					:Ton;
	tmrCartonINP					:TON;	
	tmrHorEntryPresent				:ton;
	tmrHorEntryNotPresent			:ton;	
	ServoTargetPos					:REAL;
	TimeoutTrigger					:BOOL;
	TimeoutSetting					:TIME;
	ServoMoveStarted				:BOOL;
	HOR_SpeedChange_Pos 			:REAL;
	HOR_SpeedChange_to_Exit			:BOOL;
	LightCurtain_Unmute_TON			:TON;
	bLightCurtain_Delay_Mute_Off	:BOOL;	
	CntTapeReal_SlotL				:CTU;
	CntTapeReal_SlotR				:CTU;
	FullCaseRemoved					:F_TRIG;
	Weight_reading_Dly				:Ton;
	TiltOutCv_StopDly				:Ton;
	TiltInCv_InPosDly				:TON;	
	Weight_Fail_Counter				:INT;
	
END_VAR

(**************************************************************************************************************)
(* GENERAL STATION MAPPING  *)
(**************************************************************************************************************)
Station.Name			:=	'HORIZONTAL';
Station.Rdy 			:= 	Station.Origin;
Station.AutoRun 		:=	(MC.AutoRunning OR Station.M_Step) AND 
							NOT (Station.Bypass OR Station.MajorFault OR Station.MinorFault );
Station.RunReq			:= 	(HOR_DnStream_TOFF.Q AND H_ER_CtnGlueDone)
							OR Station.M_Step;
Station.RunCond			:=	(NOT SC[6].Running OR SC[6].RunStep >= 40) AND
							NOT (Station.Done OR MC.StopPressed );
Station.Run_NextStepPls	:=	(Station.AutoRun AND NOT Station.M_Step) OR 
							(Station.M_Step AND M_StepFwdPls) OR HMI.T_OneCycleRun;
Station.Run_PrevStepPls	:=	(Station.M_Step AND M_StepBwdPls);

(**************************************************************************************************************)
(* Auto Sequance*)
(**************************************************************************************************************)

Timeout(IN:=TimeoutTrigger, PT:=TimeoutSetting);
IF Timeout.Q THEN
	TimeoutTrigger := FALSE;
END_IF

TiltOutCv_StopDly( IN:= NOT I_HOR_Tilt_Out_Cv_Present AND HOR_Tilt_Out_Mtr_Var.S_Running, PT:= T#5S); 
TiltInCv_InPosDly( IN:= I_HOR_Tilt_In_Cv_Present AND HOR_Tilt_In_Mtr_Var.S_Running, PT:= T#2S);

tmrCartonINP			(IN:=WT_Mtr_Var.S_Running AND I_HOR_Entry_Cv_Present, PT:=T#1S);
tmrHorEntryPresent		(IN:=I_HOR_Entry_Cv_Present, PT := T#100MS);
tmrHorEntryNotPresent	(IN:=NOT I_HOR_Entry_Cv_Present, PT := T#100MS);
ExitCvFull_TON			(IN:= I_HOR_DnStream_Cv_Full, pt:= T#5S);
T_ExitCvFull 			:= ExitCvFull_TON.Q AND mc.AutoMode;
W_HOR_Conv_Full			:= T_ExitCvFull;

FullCaseRemoved( CLK:= I_HOR_DnStream_Cv_Full );
IF FullCaseRemoved.Q THEN
	Exit_Case_Good 					:= FALSE;
	Exit_Case_NG					:= FALSE;
END_IF

IF E_Weigh_ConsecutiveErr AND mc.ResetPressed THEN
	Hor_Auto.Weight_Fail_Counter := 0;	
END_IF

(*********************Tape Reel turn counter *****************************)
CntTapeReal_SlotL(
	CU:= (Station.RunStep >= 20 ) AND I_HOR_TapeL_Empty_PE , 
	RESET:= Station.RunStep = 0 , 
	PV:= 3 , 
	Q=> , 
	CV=> );
	
TapeReel_ActivatedL	:= CntTapeReal_SlotL.Q;

CntTapeReal_SlotR(
	CU:= (Station.RunStep >= 20 ) AND I_HOR_TapeR_Empty_PE , 
	RESET:= Station.RunStep = 0 , 
	PV:= 3 , 
	Q=> , 
	CV=> );
	
TapeReel_ActivatedR	:= CntTapeReal_SlotR.Q;

(*-----------------------------------------------------------------------------*)

Weight_reading_Dly (IN:= Station.RunReq AND I_Weighing_Status_SteadyBit, pt:= T#0.5S);
			

IF Station.AutoRun OR Station.M_Step THEN
	
	CASE Station.RunStep OF

	0 : 	(************* Ready To Run / Capture Carton Weight ****************)
			IF 	Station.RunCond AND Station.RunReq THEN	
				TimeoutTrigger := TRUE;
				TimeoutSetting := T#30S;
			ELSE
				TimeoutTrigger := FALSE;	
			END_IF
			
			IF 	Station.RunCond AND Station.RunReq AND 
				(NOT I_HOR_DnStream_Cv_Full OR mc.DryRun) AND
				((I_Weighing_Status_SteadyBit AND	Weight_reading_Dly.q) OR
				 H_HOR_CtnWeightOK OR NOT Cfg_EnbWeightCheck OR mc.DryRun) THEN			 
				 
				IF NOT H_HOR_CtnWeightOK THEN
					H_HOR_CtnWeightOK 	:= TRUE;
					H_CartonWeight		:= DINT_TO_REAL(I_Weighing) / 1000;
				END_IF
				
				Station.RunStep 	:= Station.RunStep + 10;
				TimeoutTrigger 		:= FALSE;
			ELSIF NOT Station.RunCond THEN
				Station.Status 		:= '0: Station Waiting for Run Conditions';
				Station.StatusInt	:= 1;
			ELSIF I_HOR_DnStream_Cv_Full THEN
				Station.Status 		:= '0: Station Waiting for Exit Conveyor Empty';
				Station.StatusInt	:= 2;
			ELSIF Timeout.Q THEN
				E_Weigh_ReadingErr	:= TRUE;
			ELSE
				Station.Status 		:= '0: Station Not Ready';
				Station.StatusInt	:= 3;				
			END_IF
	

	10 : 	(************* Waiting Product Coming  ****************)
			Station.Status 		:= '20: Waiting Product Coming';
			Station.StatusInt	:= 351;
			TimeoutTrigger 		:= TRUE;
			TimeoutSetting		:= T#10S;
			
			IF Timeout.Q THEN
				E_Hor_Entry_Sensor 			:= TRUE;
			END_IF
			
				WT_Mtr_Var.In_AutoON 		:= TRUE;
				HOR_BotCv_Mtr_Var.In_AutoON := TRUE;
				HOR_TopCv_Mtr_Var.In_AutoON := TRUE;
				EX_StpCylL_Var.In_AutoHome	:= TRUE;
				EX_StpCylL_Var.In_Autowork	:= FALSE;
				EX_StpCylR_Var.In_AutoHome	:= TRUE;
				EX_StpCylR_Var.In_Autowork	:= FALSE;
				
			IF I_HOR_Entry_Cv_Present OR mc.DryRun THEN
				H_ER_CtnRdyForGlue 					:= FALSE;
				EX_FlapHoldL_Cyl_Var.In_AutoWork 	:= FALSE;
				EX_FlapHoldL_Cyl_Var.In_AutoHome 	:= TRUE;
				EX_FlapHoldR_Cyl_Var.In_AutoWork 	:= FALSE;
				EX_FlapHoldR_Cyl_Var.In_AutoHome 	:= TRUE;
				TimeoutTrigger 						:= FALSE;
				Station.RunStep	:= Station.RunStep + 10;
			END_IF
	
	20 : 	(************* Top and Bottom Conveyor Run  ****************)
			Station.Status 		:= '20: Top and Bottom Cv Run';
			Station.StatusInt	:= 352;
			HOR_BotCv_Mtr_Var.In_AutoON := TRUE;
			HOR_TopCv_Mtr_Var.In_AutoON := TRUE;
			TimeoutTrigger 		:= TRUE;
			TimeoutSetting		:= T#10S;
			(*
			IF NOT I_HOR_Entry_Cv_Present AND T_GlueEnable THEN
				EX_StpCylL_Var.In_AutoHome	:=FALSE;
				EX_StpCylL_Var.In_Autowork	:=TRUE;
				EX_StpCylR_Var.In_AutoHome	:=FALSE;
				EX_StpCylR_Var.In_Autowork	:=TRUE;
			END_IF
			*)
				EX_StpCylL_Var.In_AutoHome	:=FALSE;
				EX_StpCylL_Var.In_Autowork	:=TRUE;
				EX_StpCylR_Var.In_AutoHome	:=FALSE;
				EX_StpCylR_Var.In_Autowork	:=TRUE;
			
			IF Timeout.Q THEN
				E_Hor_Entry_Sensor := TRUE;	
			END_IF
					
			IF 	tmrHorEntryPresent.Q OR 
				mc.DryRun THEN
				WT_Mtr_Var.In_AutoON 	:= FALSE;		
				TimeoutTrigger 			:= FALSE;	
				Station.RunStep			:= Station.RunStep + 10;
			END_IF

	30 : 	(************* Carton Send to Exit Conveyor  ****************)
			Station.Status 		:= '30: Carton Send to Exit Conveyor';
			Station.StatusInt	:= 353;
			H_ER_CtnGlueDone	:= FALSE;
			TimeoutTrigger 		:= TRUE;
			TimeoutSetting		:= T#10S;
			
			IF Timeout.Q THEN
				IF NOT tmrHorEntryNotPresent.q THEN
					E_Hor_Entry_Sensor := TRUE;
				ELSIF NOT I_HOR_DnStream_Cv_Full THEN
					E_Hor_Exit_Sensor	:= TRUE;
				END_IF			
			END_IF
			
